// TwinCAT 3 PLC project PLC
// ProgramVersion: 3.1.4026.17
// CompilerDefines: VISU_USEPROPERTYINFO
// libraries:
//   Tc2_Standard, * (Beckhoff Automation GmbH)
//   Tc2_System, * (Beckhoff Automation GmbH)
//   Tc3_Analytics, * (Beckhoff Automation GmbH)
//   TcoCore, * (Vortex.Library)
//   TcoDrivesBeckhoff, * (Vortex.Library)
//   TcoElements, * (Vortex.Library)
//   TcoIo, * (Vortex.Library)
//   TcoPneumatics, * (Vortex.Library)
//   TcoUtilities, * (Vortex.Library)
//   VisuDialogs, * (System)
// project tree:
//   Components/ ST_MachineSetting.TcDUT
//   Components/TcaCarrier/Structures/ TcaCarrierConfig.TcDUT, TcaCarrierService.TcDUT, TcaCarrierData.TcDUT
//   Components/TcaCarrier/Enumerations/ eTcaCarrierCmd.TcDUT (not stored), eTcaCarrierLayout.TcDUT (not stored)
//   Components/TcaCarrier/ ITcaCarrier.TcIO, TcaCarrier.TcPOU
//   Components/TcaCarrier/Tasks/ TcaCarrierModifyTask.TcPOU
//   Components/TcaPushButton/Enumerations/ eTcaPushButtonColor.TcDUT, eTcaPushButtonLightState.TcDUT
//   Components/TcaPushButton/Structures/ TcaPushButtonStatus.TcDUT (not stored), TcaPushButtonRef.TcDUT (not stored), TcaPushButtonConfig.TcDUT (not stored), TcaPushButtonService.TcDUT
//   Components/TcaPushButton/ TcaPushButton.TcPOU
//   Components/TcaStorage/ E_ApproachDirection.TcDUT (not stored), eTcaStorageCmd.TcDUT, TcaRobotStorage.TcPOU (not stored) (excluded from build), TcaStorage.TcPOU, TcaStorageRef.TcDUT
//   Components/TcaTrolley/Structures/ TcaTrolleyData.TcDUT, TcaTrolleyService.TcDUT
//   Components/TcaTrolley/ TcaTrolley.TcPOU
//   Components/TcaTrolley_old/ CMD_Trolley.TcDUT, eTcaTrolleyCmd.TcDUT (not stored), TcaTrolley_old.TcPOU, TcaTrolleyRef.TcDUT (not stored)
//   Components/TcaWorkpiecePlace/Enumerations/ eTcaWorkpiecePlaceStatus.TcDUT, eTcaWorkpiecePlaceShape.TcDUT
//   Components/TcaWorkpiecePlace/Structures/ TcaWorkpiecePlaceService.TcDUT, TcaWorkpiecePlaceData.TcDUT
//   Components/TcaWorkpiecePlace/ TcaWorkpiecePlace.TcPOU
//   Components_RMTH/TcaEngelCasting/ Schnittstellenprotokoll.TcDUT (not stored), TcaEngelCastingCarrierInput.TcDUT (not stored), TcaEngelCastingCarrierJob.TcDUT (not stored), TcaEngelCastingCarrierJobStatus.TcDUT, TcaEngelCastingCarrierOutput.TcDUT (not stored), TcalEngelCastingCarrierStatus.TcDUT (not stored)
//   Components_RMTH/TcaLaserDistanceSenor/Structures/ TcaLaserDistanceSenorConfig.TcDUT (not stored), TcaLaserDistanceSenorRef.TcDUT (not stored), TcaLaserDistanceSenorStatus.TcDUT, TcaLaserDistanceSensorDataArrayEntry.TcDUT (not stored), TcaLaserDistanceSenorService.TcDUT (not stored)
//   Components_RMTH/TcaLaserDistanceSenor/ TcaLaserDistanceSenor.TcPOU (not stored)
//   Components_RMTH/TcaRackFeeder/Structures/ TcaRackFeederConfig.TcDUT (not stored), TcaRackFeederRef.TcDUT (not stored), TcaRackFeederService.TcDUT (not stored), TcaRackFeederStatus.TcDUT
//   Components_RMTH/TcaRackFeeder/ TcaRackFeeder.TcPOU (not stored)
//   Components_RMTH/TcaSafetyGate/ ISafetyComponent.TcIO (not stored), TcaSafetyGate.TcPOU (not stored)
//   Components_RMTH/TcaSafetyGate/Structures/ TcaSafetyGateConfig.TcDUT (not stored), TcaSafetyGateRef.TcDUT, TcaSafetyGateService.TcDUT, TcaSafetyGateStatus.TcDUT
//   Components_RMTH/TcaSegmentDoor/Structures/ TcaSegmentDoorConfig.TcDUT (not stored), TcaSegmentDoorRef.TcDUT (not stored), TcaSegmentDoorService.TcDUT (not stored), TcaSegmentDoorStatus.TcDUT (not stored)
//   Components_RMTH/TcaSegmentDoor/ TcaSegmentDoor.TcPOU
//   Components_RMTH/TcaTwinSAFE/Structures/ TcaTwinSAFEConfig.TcDUT, TcaTwinSAFERef.TcDUT (not stored), TcaTwinSAFEService.TcDUT (not stored), TcaTwinSAFEStatus.TcDUT (not stored)
//   Components_RMTH/TcaTwinSAFE/ TcaTwinSAFE.TcPOU (not stored)
//   / GlobalTextList.TcGTLO, PlcTask.TcTTO, Visualization Manager.TcVMO (not stored)
//   Items/ COLOR.TcDUT, E_Coordinate.TcDUT (not stored), ST_ComboboxEntry.TcDUT, ST_Coordinate.TcDUT (not stored), ST_WorkpieceType.TcDUT
//   Program/Handling/Dialogs/ Handling_TeachRack_DlgContent.TcPOU
//   Program/Handling/Sequences/ Handling_Teach.TcPOU (not stored), Handling_TeachRack.TcPOU (not stored), Handling_GroundMode.TcPOU (not stored), Handling_OpenDoor.TcPOU (not stored)
//   Program/ MAIN.TcPOU, Peripherie.TcPOU
//   Program/Handling/ Handling.TcPOU, Handling_Components.TcPOU (not stored), Handling_Positions.TcPOU (not stored)
//   Template/Component_Cylinder/Base/ CylinderBase.TcPOU, TcoCylinderBase.TcPOU (not stored), TcoDoubleCylinderBase.TcPOU
//   Template/Component_Cylinder/ ITcoCylinder.TcIO (not stored), TcoCylinder.TcPOU, TcoDoubleCylinder.TcPOU
//   Template/Component_Cylinder/Structs/ CylinderConfig.TcDUT, CylinderStatus.TcDUT (not stored), TcoCylinderConfig.TcDUT, TcoCylinderStatus.TcDUT
//   Template/Component_Cylinder/Tasks/ CylinderMoveTask.TcPOU, TcoCylinderMoveTask.TcPOU (not stored)
//   Template/RackFeeder/ CMD_RackFeeder.TcDUT, E_RackFeederCmd.TcDUT (not stored), FB_RackFeeder.TcPOU
//   Template/RackFeeder/Structure/ ST_RackFeederIO.TcDUT, ST_RackFeederJob.TcDUT (not stored), ST_StorageDock.TcDUT (not stored), ST_TrolleyDock.TcDUT (not stored)
//   Template/Station/Data/ ST001_ProcessData.TcDUT (not stored), ST001_ProcessDataManager.TcPOU (not stored)
//   Template/Station/ ST001.TcPOU, ST001_AutomatSequence.TcPOU (not stored), ST001_Components.TcDUT (not stored), ST001_ComponentsHandler.TcPOU, ST001_GroundSequence.TcPOU
//   Template/Component_Carousell/Base/ TcoCarouselBase.TcPOU (not stored)
//   Template/Component_Carousell/Structs/ eTcoCarouselDirection.TcDUT, TcoCarouselConfig.TcDUT, TcoCarouselStatus.TcDUT
//   Template/Component_Carousell/Tasks/ TcoTurnTableTask.TcPOU
//   Template/Component_Carousell/ TcoCarousel.TcPOU (not stored)
//   Utilities/Component/Enumerations/ E_ComponentState.TcDUT, E_SafeState.TcDUT (not stored)
//   Utilities/Component/ FB_Component.TcPOU, FB_ComponentPool.TcPOU (not stored)
//   Utilities/Component/Interfaces/ ITF_Component.TcIO (not stored)
//   Utilities/Component/Structures/ ST_ComponentVisu.TcDUT
//   Utilities/Component/Visualisation/ Uc_Component.TcVIS (not stored)
//   Utilities/EventLog/Base/ FB_LoggingProviderBase.TcPOU (not stored)
//   Utilities/EventLog/Enumerations/ E_BoolFilter.TcDUT (not stored), E_FilterActive.TcDUT (not stored), E_LoggingProvider.TcDUT, E_LogLevel.TcDUT (not stored), E_Priority.TcDUT, ST_LoggingConfig.TcDUT (not stored)
//   Utilities/EventLog/ E_Event.TcDUT, FB_EventLog.TcPOU
//   Utilities/EventLog/Interface/ ITFLoggingProvider.TcIO, ITF_EventLog.TcIO (not stored)
//   Utilities/EventLog/Structures/ ST_Event.TcDUT (not stored), ST_EventBase.TcDUT, ST_EventOutput.TcDUT (not stored), ST_EventVisu.TcDUT, ST_Log.TcDUT (not stored)
//   Utilities/EventLog/Visualization/ Uc_EventLog.TcVIS (not stored), Uc_EventLogControl.TcDUT (not stored), Uc_EventLogControl.TcVIS (not stored), Uc_EventLogEntry.TcVIS (not stored), Uc_EventLogTable.TcDUT (not stored), Uc_EventLogTable.TcVIS (not stored)
//   Utilities/Helpers/Color/ F_DWORD2CMYK.TcPOU (not stored), F_DWORD2RGB.TcPOU, F_RGB2CMYK.TcPOU, F_RGB2DWORD.TcPOU (not stored), F_TextColor.TcPOU, ST_Color.TcDUT (not stored), ST_ColorCMYK.TcDUT
//   Utilities/Helpers/Concat/ Concat10.TcPOU (not stored), Concat2.TcPOU, Concat3.TcPOU (not stored), Concat4.TcPOU (not stored), Concat5.TcPOU (not stored), Concat6.TcPOU (not stored), Concat7.TcPOU, Concat8.TcPOU (not stored), Concat9.TcPOU (not stored), ConcatArray.TcPOU (not stored)
//   Utilities/Helpers/ E_OperationResult.TcDUT, FB_GetTimeString.TcPOU (not stored) (excluded from build), FB_Pulse.TcPOU (not stored), FB_TON_RMTH.TcPOU (not stored), F_BYTE_TO_INT.TcPOU (not stored), F_BYTE_TO_REAL.TcPOU, F_DT_TO_STRING.TcPOU, F_GetAdsPort.TcPOU, F_GetPlcCycleTime.TcPOU (not stored), F_GetSystemTime64.TcPOU (not stored), F_TO_STRING.TcPOU (not stored), P_FilePath.TcPOU, P_System.TcPOU (not stored), ST_DefaultPulse.TcDUT, ST_PlcSystemInfo.TcDUT
//   Utilities/ HexColor.TcGVL (not stored), Statics.TcGVL (not stored), StaticsConstant.TcGVL
//   Utilities/List/ FB_List.TcPOU
//   Utilities/List/Structures/ ST_Listentry.TcDUT, Uc_List.TcDUT (not stored)
//   Utilities/List/Visu/ Uc_EntryDetail.TcVIS, Uc_List.TcVIS (not stored), Uc_Listentry.TcVIS (not stored)
//   Utilities/Sequencer/Enumeration/ E_SequenceState.TcDUT (not stored)
//   Utilities/Sequencer/ FB_Sequence.TcPOU (not stored)
// real-time tasks:
//   TASK PlcTask: cycle T#10ms, priority 20, ADS port 350
// motion (NC):
//   TASK NC-Task 1 SAF: cycle T#2ms, priority 4, ADS port 501
//   TASK NC-Task 1 SVB: cycle T#10ms, priority 8, ADS port 511
//   AXIS Oven B CH1 (id 14)
//     Dynamic: Acceleration=282800000, Deceleration=282800000, Jerk=2.85628e+17
//     Velo: RefSearch=25, RefSync=25, SlowManual=14, FastManual=28, Maximum=28
//     PositionAreaControl: Enable=false
//     TargetPosControl: Enable=false
//     OtherSettings: AllowMotionCmdToSlave=true
//     encoder EncType=7
//       EncPara: ScaleFactorNumerator=0.001879, Offset=-1.4, MaxCount=#x0000ffff, ReferenceSystem=1
//     drive DrvType=23
//       Analog: VeloReferenz=28, TorqueSetpointScale=10, ScaleFactorActTorque=0.1
//       TimeComp: TaskDelayCycles=1
//     controller CtrType=1
//       CtrPara: PriorControlFactor=1
//         PosDiffControl: Enable=false
//         Observer: BandWidth=20
//   AXIS Storage A (id 2)
//     Dynamic: Acceleration=282800000, Deceleration=282800000, Jerk=2.85628e+17
//     Velo: RefSearch=25, RefSync=25, SlowManual=14, FastManual=28, Maximum=28
//     PositionAreaControl: Enable=false
//     TargetPosControl: Enable=false
//     OtherSettings: AllowMotionCmdToSlave=true
//     encoder EncType=1
//       EncPara: ScaleFactorNumerator=0.00751766651631334, Offset=-1.4
//     drive DrvType=23
//       Analog: VeloReferenz=28, TorqueSetpointScale=10, ScaleFactorActTorque=0.1
//       TimeComp: TaskDelayCycles=1
//     controller CtrType=1
//       CtrPara: PriorControlFactor=1
//         PosDiffControl: Enable=false
//         Observer: BandWidth=20
//   AXIS Oven B CH2 (id 15)
//     Dynamic: Acceleration=282800000, Deceleration=282800000, Jerk=2.85628e+17
//     Velo: RefSearch=25, RefSync=25, SlowManual=14, FastManual=28, Maximum=28
//     PositionAreaControl: Enable=false
//     TargetPosControl: Enable=false
//     OtherSettings: AllowMotionCmdToSlave=true
//     encoder EncType=7
//       EncPara: ScaleFactorNumerator=0.001879, Offset=-1.4, MaxCount=#x0000ffff, ReferenceSystem=1
//     drive DrvType=23
//       Analog: VeloReferenz=28, TorqueSetpointScale=10, ScaleFactorActTorque=0.1
//       TimeComp: TaskDelayCycles=1
//     controller CtrType=1
//       CtrPara: PriorControlFactor=1
//         PosDiffControl: Enable=false
//         Observer: BandWidth=20
//   AXIS Rackfeeder X (id 16)
//     Dynamic: Acceleration=2461.9275, Deceleration=2461.9275, Jerk=7385.7825
//     Velo: RefSearch=16.41285, RefSync=16.41285, SlowManual=10, FastManual=60, Fast=1641.285, Maximum=1641.285
//     OtherSettings: AllowMotionCmdToSlave=true
//     encoder EncType=8
//       EncPara: ScaleFactorNumerator=150, ScaleFactorDenominator=10485760, MaxCount=#xffffffff
//     drive DrvType=9
//       DrvPara: MaxCount=#xffffffff, DriveControlDWord=#x00030100
//         Analog: VeloReferenz=1805.4135, VeloScale=1.02400649589962, TorqueSetpointScale=10, ScaleFactorActTorque=0.1
//         TimeComp: TaskDelayCycles=1
//     controller CtrType=1
//       CtrPara: PriorControlFactor=1
//         Observer: BandWidth=20
//   AXIS Rackfeeder Y (id 17)
//     Dynamic: Acceleration=2256.7665, Deceleration=2256.7665, Jerk=6770.2995
//     Velo: RefSearch=15.04511, RefSync=15.04511, SlowManual=10, FastManual=60, Fast=1504.511, Maximum=1504.511
//     OtherSettings: AllowMotionCmdToSlave=true
//     encoder EncType=8
//       EncPara: ScaleFactorNumerator=220, ScaleFactorDenominator=16777216, MaxCount=#xffffffff
//     drive DrvType=9
//       DrvPara: MaxCount=#xffffffff, DriveControlDWord=#x00030100
//         Analog: VeloReferenz=1654.9621, VeloScale=1.02400649589962, TorqueSetpointScale=10, ScaleFactorActTorque=0.1
//         TimeComp: TaskDelayCycles=1
//     controller CtrType=1
//       CtrPara: PriorControlFactor=1
//         Observer: BandWidth=20
//   AXIS Rackfeeder Teleskop (id 18)
//     OtherSettings: AllowMotionCmdToSlave=true
//     encoder EncType=8
//       EncPara: MaxCount=#xffffffff
//     drive DrvType=9
//       DrvPara: MaxCount=#xffffffff, DriveControlDWord=#x00030100
//         Analog: VeloScale=1.02400649589962, TorqueSetpointScale=10, ScaleFactorActTorque=0.1
//         TimeComp: TaskDelayCycles=1
//     controller CtrType=1
//       CtrPara: PriorControlFactor=1
//         Observer: BandWidth=20
//   AXIS Oven B (id 21)
//     Dynamic: Acceleration=1231.0125, Deceleration=1231.0125, Jerk=3693.0375
//     Velo: RefSearch=8.20675, RefSync=8.20675, SlowManual=20, FastManual=120, Fast=820.675, Maximum=820.675
//     OtherSettings: AllowMotionCmdToSlave=true
//     encoder EncType=8
//       EncPara: ScaleFactorNumerator=120, ScaleFactorDenominator=16777216, Inverse=true, MaxCount=#xffffffff
//     drive DrvType=9
//       DrvPara: Inverse=true, MaxCount=#xffffffff, DriveControlDWord=#x00030100
//         Analog: VeloReferenz=902.7425, VeloScale=1.02400649589962, TorqueSetpointScale=10, ScaleFactorActTorque=0.1
//         TimeComp: TaskDelayCycles=1
//     controller CtrType=1
//       CtrPara: PriorControlFactor=1
//         Observer: BandWidth=20
//   AXIS Oven A (id 20)
//     Dynamic: Acceleration=1231.0125, Deceleration=1231.0125, Jerk=3693.0375
//     Velo: RefSearch=8.20675, RefSync=8.20675, SlowManual=20, FastManual=120, Fast=820.675, Maximum=820.675
//     OtherSettings: AllowMotionCmdToSlave=true
//     encoder EncType=8
//       EncPara: ScaleFactorNumerator=120, ScaleFactorDenominator=16777216, Inverse=true, MaxCount=#xffffffff
//     drive DrvType=9
//       DrvPara: Inverse=true, MaxCount=#xffffffff, DriveControlDWord=#x00030100
//         Analog: VeloReferenz=902.7425, VeloScale=1.02400649589962, TorqueSetpointScale=10, ScaleFactorActTorque=0.1
//         TimeComp: TaskDelayCycles=1
//     controller CtrType=1
//       CtrPara: PriorControlFactor=1
//         Observer: BandWidth=20
//   AXIS Oven A CH1 (id 1)
//     Dynamic: Acceleration=282800000, Deceleration=282800000, Jerk=2.85628e+17, DelayTime=0.01, OverrideType=4
//     Velo: RefSearch=25, RefSync=25, SlowManual=14, FastManual=28, Maximum=28
//     PositionAreaControl: Enable=false
//     TargetPosControl: Enable=false
//     OtherSettings: AllowMotionCmdToSlave=true
//     encoder EncType=7
//       EncPara: ScaleFactorNumerator=0.001879, Offset=-1.4, EncMode=1, MaxCount=#x0000ffff, ReferenceSystem=1
//         FilterTime: TVelo=0.1
//         SoftEndMinControl: Range=-5
//         SoftEndMaxControl: Range=30
//         ActPosCorrection: Enable=true, Time=1
//     drive DrvType=23
//       Analog: VeloReferenz=28, TorqueSetpointScale=10, ScaleFactorActTorque=0.1
//       TimeComp: TaskDelayCycles=1
//     controller CtrType=1
//       CtrPara: PriorControlFactor=1
//         PosDiffControl: Enable=false
//         Observer: BandWidth=20
//   AXIS Oven A CH2 (id 13)
//     Dynamic: Acceleration=282800000, Deceleration=282800000, Jerk=2.85628e+17
//     Velo: RefSearch=25, RefSync=25, SlowManual=14, FastManual=28, Maximum=28
//     PositionAreaControl: Enable=false
//     TargetPosControl: Enable=false
//     OtherSettings: AllowMotionCmdToSlave=true
//     encoder EncType=7
//       EncPara: ScaleFactorNumerator=0.001879, Offset=-1.4, MaxCount=#x0000ffff, ReferenceSystem=1
//     drive DrvType=23
//       Analog: VeloReferenz=28, TorqueSetpointScale=10, ScaleFactorActTorque=0.1
//       TimeComp: TaskDelayCycles=1
//     controller CtrType=1
//       CtrPara: PriorControlFactor=1
//         PosDiffControl: Enable=false
//         Observer: BandWidth=20
//   AXIS Storage B (id 3)
//     Dynamic: Acceleration=282800000, Deceleration=282800000, Jerk=2.85628e+17
//     Velo: RefSearch=25, RefSync=25, SlowManual=14, FastManual=28, Maximum=28
//     PositionAreaControl: Enable=false
//     TargetPosControl: Enable=false
//     OtherSettings: AllowMotionCmdToSlave=true
//     encoder EncType=1
//       EncPara: ScaleFactorNumerator=0.00751766651631334, Offset=-1.4
//     drive DrvType=23
//       Analog: VeloReferenz=28, TorqueSetpointScale=10, ScaleFactorActTorque=0.1
//       TimeComp: TaskDelayCycles=1
//     controller CtrType=1
//       CtrPara: PriorControlFactor=1
//         PosDiffControl: Enable=false
//         Observer: BandWidth=20
// I/O:
//   DEVICE Gerät 3 (EtherCAT) (disabled), AmsNetId 41.249.230.93.4.1
//     Klemme 1 (EK1100) [EK1100 EtherCAT-Koppler (2A E-Bus)]
//       Klemme 33 (EL6910) [EL6910, TwinSAFE PLC]
//       Klemme 3 (EL1904) [EL1904, 4 K. Safety Eingang 24V, TwinSAFE]
//         modules: Module 1 (FSOES)
//       Klemme 4 (EL2904) [EL2904, 4 K. Safety Ausgang 24V, 0.5A, TwinSAFE]
//         modules: Module 1 (FSOES), Module 2 (DO)
//       Klemme 5 (EL1104) [EL1104 4K. Dig. Eingang 24V, 3ms, Sensorversorgung]
//       Klemme 6 (EL1104) [EL1104 4K. Dig. Eingang 24V, 3ms, Sensorversorgung]
//       Klemme 7 (EL6224) [EL6224 (IO Link Master)]
//       ENGEL Interface (EL1008) [EL1008 8K. Dig. Eingang 24V, 3ms]
//       ENGEL Interface (EL2624) [EL2624 4K. Relais Ausgang, Schließer (125V AC / 30V DC)]
//       Ovens (EK1122) [EK1122 2-Port EtherCAT-Abzweig]
//         Oven_A (EK1100) [EK1100 EtherCAT-Koppler (2A E-Bus)]
//           Klemme 10 (EL1904) [EL1904, 4 K. Safety Eingang 24V, TwinSAFE]
//             modules: Module 1 (FSOES)
//           Klemme 11 (EL2904) [EL2904, 4 K. Safety Ausgang 24V, 0.5A, TwinSAFE]
//             modules: Module 1 (FSOES), Module 2 (DO)
//           Klemme 12 (EL7332) [EL7332 2K. DC-Motor-Endstufe (24V, 1.5A)]
//           Klemme 13 (EL3062-0030) [EL3062-0030 2K.Ana. Eingang 0-30V]
//           Klemme 14 (EL1004) [EL1004 4K. Dig. Eingang 24V, 3ms]
//           Klemme 15 (EL2004) [EL2004 4K. Dig. Ausgang 24V, 0.5A]
//           Klemme 16 (EL9010) [EL9010 Endklemme]
//         Oven_B (EK1100) [EK1100 EtherCAT-Koppler (2A E-Bus)]
//           Klemme 18 (EL1904) [EL1904, 4 K. Safety Eingang 24V, TwinSAFE]
//             modules: Module 1 (FSOES)
//           Klemme 19 (EL2904) [EL2904, 4 K. Safety Ausgang 24V, 0.5A, TwinSAFE]
//             modules: Module 1 (FSOES), Module 2 (DO)
//           Klemme 20 (EL7332) [EL7332 2K. DC-Motor-Endstufe (24V, 1.5A)]
//           Klemme 21 (EL3062-0030) [EL3062-0030 2K.Ana. Eingang 0-30V]
//           Klemme 22 (EL1004) [EL1004 4K. Dig. Eingang 24V, 3ms]
//           Klemme 23 (EL2004) [EL2004 4K. Dig. Ausgang 24V, 0.5A]
//           Klemme 61 (EL9010) [EL9010 Endklemme]
//       Storage|Casting (EK1122) [EK1122 2-Port EtherCAT-Abzweig]
//         Storage (EK1100)
//     RackFeeder_X_Y (AX5206-0000-0215) [AX5206-0000-0215 EtherCAT Drive (SoE, 2 Ch.)]
//       Klemme 27 (AX5805) [AX5805 (Safety Drive Option)]
//         modules: Module 1 (Safety Process Data, 2 axis), Module 2 (Standard Process Data, 2 axis)
//     Rackfeeder_Teleskop (AX5203-0000-0215) [AX5203-0000-0215 EtherCAT Drive (SoE, 2 Ch.)]
//       Klemme 29 (AX5805) [AX5805 (Safety Drive Option)]
//         modules: Module 1 (Safety Process Data, 2 axis), Module 2 (Standard Process Data, 2 axis)
//     OvenDoor_A_B (AX5206-0000-0215) [AX5206-0000-0215 EtherCAT Drive (SoE, 2 Ch.)]
//       Klemme 31 (AX5805) [AX5805 (Safety Drive Option)]
//         modules: Module 1 (Safety Process Data, 2 axis), Module 2 (Standard Process Data, 2 axis)
// variable links:
//   Device 3 (EtherCAT) <-> Device 3 (EtherCAT)/OvenDoor_A_B (AX5206-0000-0215)/Term 31 (AX5805)
//     Term 1 (EK1100)/Term 33 (EL6910)/ConnectionInputs/TwinSafeMain.Oven (AX5805) - Module 1 (Safety Process Data, 2 axis)_120 TxPDO <-> Module 1 (Safety Process Data, 2 axis)/Outputs (Controlword)/FSOE
//     Term 1 (EK1100)/Term 33 (EL6910)/ConnectionOutputs/TwinSafeMain.Oven (AX5805) - Module 1 (Safety Process Data, 2 axis)_120 RxPDO <-> Module 1 (Safety Process Data, 2 axis)/Inputs (Statusword)/FSOE
//   Device 3 (EtherCAT) <-> Device 3 (EtherCAT)/RackFeeder_X_Y (AX5206-0000-0215)/Term 27 (AX5805)
//     Term 1 (EK1100)/Term 33 (EL6910)/ConnectionInputs/TwinSafeMain.Rackfeeder_XY (AX5805) - Module 1 (Safety Process Data, 2 axis)_118 TxPDO <-> Module 1 (Safety Process Data, 2 axis)/Outputs (Controlword)/FSOE
//     Term 1 (EK1100)/Term 33 (EL6910)/ConnectionOutputs/TwinSafeMain.Rackfeeder_XY (AX5805) - Module 1 (Safety Process Data, 2 axis)_118 RxPDO <-> Module 1 (Safety Process Data, 2 axis)/Inputs (Statusword)/FSOE
//   Device 3 (EtherCAT) <-> Device 3 (EtherCAT)/Rackfeeder_Teleskop (AX5203-0000-0215)/Term 29 (AX5805)
//     Term 1 (EK1100)/Term 33 (EL6910)/ConnectionInputs/TwinSafeMain.Rackfeeder_Tele (AX5805) - Module 1 (Safety Process Data, 2 axis)_119 TxPDO <-> Module 1 (Safety Process Data, 2 axis)/Outputs (Controlword)/FSOE
//     Term 1 (EK1100)/Term 33 (EL6910)/ConnectionOutputs/TwinSafeMain.Rackfeeder_Tele (AX5805) - Module 1 (Safety Process Data, 2 axis)_119 RxPDO <-> Module 1 (Safety Process Data, 2 axis)/Inputs (Statusword)/FSOE
//   Device 3 (EtherCAT) <-> Device 3 (EtherCAT)/Term 1 (EK1100)/Ovens (EK1122)/Oven_A (EK1100)/Term 10 (EL1904)
//     Term 1 (EK1100)/Term 33 (EL6910)/ConnectionInputs/TwinSafeMain.Oven A (EL1904) - Module 1 (FSOES)_14 TxPDO <-> Module 1 (FSOES)/RxPDO/FSOE
//     Term 1 (EK1100)/Term 33 (EL6910)/ConnectionOutputs/TwinSafeMain.Oven A (EL1904) - Module 1 (FSOES)_14 RxPDO <-> Module 1 (FSOES)/TxPDO/FSOE
//   Device 3 (EtherCAT) <-> Device 3 (EtherCAT)/Term 1 (EK1100)/Ovens (EK1122)/Oven_A (EK1100)/Term 11 (EL2904)
//     Term 1 (EK1100)/Term 33 (EL6910)/ConnectionInputs/TwinSafeMain.Oven A (EL2904) - Module 1 (FSOES)_111 TxPDO <-> Module 1 (FSOES)/RxPDO/FSOE
//     Term 1 (EK1100)/Term 33 (EL6910)/ConnectionOutputs/TwinSafeMain.Oven A (EL2904) - Module 1 (FSOES)_111 RxPDO <-> Module 1 (FSOES)/TxPDO/FSOE
//   Device 3 (EtherCAT) <-> Device 3 (EtherCAT)/Term 1 (EK1100)/Ovens (EK1122)/Oven_B (EK1100)/Term 18 (EL1904)
//     Term 1 (EK1100)/Term 33 (EL6910)/ConnectionInputs/TwinSafeMain.Oven B (EL1904) - Module 1 (FSOES)_16 TxPDO <-> Module 1 (FSOES)/RxPDO/FSOE
//     Term 1 (EK1100)/Term 33 (EL6910)/ConnectionOutputs/TwinSafeMain.Oven B (EL1904) - Module 1 (FSOES)_16 RxPDO <-> Module 1 (FSOES)/TxPDO/FSOE
//   Device 3 (EtherCAT) <-> Device 3 (EtherCAT)/Term 1 (EK1100)/Ovens (EK1122)/Oven_B (EK1100)/Term 19 (EL2904)
//     Term 1 (EK1100)/Term 33 (EL6910)/ConnectionInputs/TwinSafeMain.Oven B (EL2904) - Module 1 (FSOES)_112 TxPDO <-> Module 1 (FSOES)/RxPDO/FSOE
//     Term 1 (EK1100)/Term 33 (EL6910)/ConnectionOutputs/TwinSafeMain.Oven B (EL2904) - Module 1 (FSOES)_112 RxPDO <-> Module 1 (FSOES)/TxPDO/FSOE
//   Device 3 (EtherCAT) <-> Device 3 (EtherCAT)/Term 1 (EK1100)/Term 3 (EL1904)
//     Term 1 (EK1100)/Term 33 (EL6910)/ConnectionInputs/TwinSafeMain.MAIN (EL1904) - Module 1 (FSOES)_12 TxPDO <-> Module 1 (FSOES)/RxPDO/FSOE
//     Term 1 (EK1100)/Term 33 (EL6910)/ConnectionOutputs/TwinSafeMain.MAIN (EL1904) - Module 1 (FSOES)_12 RxPDO <-> Module 1 (FSOES)/TxPDO/FSOE
//   Device 3 (EtherCAT) <-> Device 3 (EtherCAT)/Term 1 (EK1100)/Term 4 (EL2904)
//     Term 1 (EK1100)/Term 33 (EL6910)/ConnectionInputs/TwinSafeMain.MAIN (EL2904) - Module 1 (FSOES)_13 TxPDO <-> Module 1 (FSOES)/RxPDO/FSOE
//     Term 1 (EK1100)/Term 33 (EL6910)/ConnectionOutputs/TwinSafeMain.MAIN (EL2904) - Module 1 (FSOES)_13 RxPDO <-> Module 1 (FSOES)/TxPDO/FSOE
//   NC-Task 1 SAF/Axes/Oven A <-> Device 3 (EtherCAT)/OvenDoor_A_B (AX5206-0000-0215)
//     Drive/Inputs/In/nDataIn1 <-> AT 1/Following distance
//     Drive/Inputs/In/nDcOutputTime <-> InfoData/DcOutputShift
//     Drive/Inputs/In/nState1 <-> AT 1/Drive status word @bit 8
//     Drive/Inputs/In/nState2 <-> AT 1/Drive status word
//     Drive/Inputs/In/nState4 @bit 1 <-> WcState/InputToggle
//     Drive/Inputs/In/nState4 <-> WcState/WcState
//     Drive/Outputs/Out/nCtrl1 <-> MDT 1/Master control word @bit 8
//     Drive/Outputs/Out/nDataOut1 <-> MDT 1/Position command value
//     Enc/Inputs/In/nDataIn1 <-> AT 1/Position feedback 1 value
//     Enc/Inputs/In/nDcInputTime <-> InfoData/DcInputShift
//     Enc/Inputs/In/nState4 @bit 1 <-> WcState/InputToggle
//     Enc/Inputs/In/nState4 <-> WcState/WcState
//   NC-Task 1 SAF/Axes/Oven A CH1 <-> Device 3 (EtherCAT)/Term 1 (EK1100)/Ovens (EK1122)/Oven_A (EK1100)/Term 12 (EL7332)
//     Drive/Inputs/In/nState1 @bit 3 <-> DCM Status Channel 1/Status/Error
//     Drive/Inputs/In/nState1 @bit 5 <-> DCM Status Channel 1/Status/Moving negative
//     Drive/Inputs/In/nState1 @bit 4 <-> DCM Status Channel 1/Status/Moving positive
//     Drive/Inputs/In/nState1 @bit 1 <-> DCM Status Channel 1/Status/Ready
//     Drive/Inputs/In/nState1 <-> DCM Status Channel 1/Status/Ready to enable
//     Drive/Inputs/In/nState1 @bit 6 <-> DCM Status Channel 1/Status/Torque reduced
//     Drive/Inputs/In/nState1 @bit 2 <-> DCM Status Channel 1/Status/Warning
//     Drive/Inputs/In/nState2 @bit 3 <-> DCM Status Channel 1/Status/Digital input 1
//     Drive/Inputs/In/nState2 @bit 4 <-> DCM Status Channel 1/Status/Digital input 2
//     Drive/Inputs/In/nState2 @bit 5 <-> DCM Status Channel 1/Status/Sync error
//     Drive/Inputs/In/nState2 @bit 7 <-> DCM Status Channel 1/Status/TxPDO Toggle
//     Drive/Inputs/In/nState4 @bit 1 <-> WcState/InputToggle
//     Drive/Inputs/In/nState4 <-> WcState/WcState
//     Drive/Outputs/Out/nCtrl1 <-> DCM Control Channel 1/Control/Enable
//     Drive/Outputs/Out/nCtrl1 @bit 2 <-> DCM Control Channel 1/Control/Reduce torque
//     Drive/Outputs/Out/nCtrl1 @bit 1 <-> DCM Control Channel 1/Control/Reset
//     Drive/Outputs/Out/nDataOut2[0] <-> DCM Velocity Channel 1/Velocity
//   NC-Task 1 SAF/Axes/Oven A CH1 <-> Device 3 (EtherCAT)/Term 1 (EK1100)/Ovens (EK1122)/Oven_A (EK1100)/Term 13 (EL3062-0030)
//     Enc/Inputs/In/nDataIn1[0] <-> AI Standard Channel 1/Value
//     Enc/Inputs/In/nState4 @bit 1 <-> WcState/InputToggle
//     Enc/Inputs/In/nState4 <-> WcState/WcState
//   NC-Task 1 SAF/Axes/Oven A CH2 <-> Device 3 (EtherCAT)/Term 1 (EK1100)/Ovens (EK1122)/Oven_A (EK1100)/Term 12 (EL7332)
//     Drive/Inputs/In/nState1 @bit 3 <-> DCM Status Channel 2/Status/Error
//     Drive/Inputs/In/nState1 @bit 5 <-> DCM Status Channel 2/Status/Moving negative
//     Drive/Inputs/In/nState1 @bit 4 <-> DCM Status Channel 2/Status/Moving positive
//     Drive/Inputs/In/nState1 @bit 1 <-> DCM Status Channel 2/Status/Ready
//     Drive/Inputs/In/nState1 <-> DCM Status Channel 2/Status/Ready to enable
//     Drive/Inputs/In/nState1 @bit 6 <-> DCM Status Channel 2/Status/Torque reduced
//     Drive/Inputs/In/nState1 @bit 2 <-> DCM Status Channel 2/Status/Warning
//     Drive/Inputs/In/nState2 @bit 3 <-> DCM Status Channel 2/Status/Digital input 1
//     Drive/Inputs/In/nState2 @bit 4 <-> DCM Status Channel 2/Status/Digital input 2
//     Drive/Inputs/In/nState2 @bit 5 <-> DCM Status Channel 2/Status/Sync error
//     Drive/Inputs/In/nState2 @bit 7 <-> DCM Status Channel 2/Status/TxPDO Toggle
//     Drive/Inputs/In/nState4 @bit 1 <-> WcState/InputToggle
//     Drive/Inputs/In/nState4 <-> WcState/WcState
//     Drive/Outputs/Out/nCtrl1 <-> DCM Control Channel 2/Control/Enable
//     Drive/Outputs/Out/nCtrl1 @bit 2 <-> DCM Control Channel 2/Control/Reduce torque
//     Drive/Outputs/Out/nCtrl1 @bit 1 <-> DCM Control Channel 2/Control/Reset
//     Drive/Outputs/Out/nDataOut2[0] <-> DCM Velocity Channel 2/Velocity
//   NC-Task 1 SAF/Axes/Oven A CH2 <-> Device 3 (EtherCAT)/Term 1 (EK1100)/Ovens (EK1122)/Oven_A (EK1100)/Term 13 (EL3062-0030)
//     Enc/Inputs/In/nDataIn1[0] <-> AI Standard Channel 2/Value
//     Enc/Inputs/In/nState4 @bit 1 <-> WcState/InputToggle
//     Enc/Inputs/In/nState4 <-> WcState/WcState
//   NC-Task 1 SAF/Axes/Oven B <-> Device 3 (EtherCAT)/OvenDoor_A_B (AX5206-0000-0215)
//     Drive/Inputs/In/nDataIn1 <-> AT 2/Following distance
//     Drive/Inputs/In/nDcOutputTime <-> InfoData/DcOutputShift
//     Drive/Inputs/In/nState1 <-> AT 2/Drive status word @bit 8
//     Drive/Inputs/In/nState2 <-> AT 2/Drive status word
//     Drive/Inputs/In/nState4 @bit 1 <-> WcState/InputToggle
//     Drive/Inputs/In/nState4 <-> WcState/WcState
//     Drive/Outputs/Out/nCtrl1 <-> MDT 2/Master control word @bit 8
//     Drive/Outputs/Out/nDataOut1 <-> MDT 2/Position command value
//     Enc/Inputs/In/nDataIn1 <-> AT 2/Position feedback 1 value
//     Enc/Inputs/In/nDcInputTime <-> InfoData/DcInputShift
//     Enc/Inputs/In/nState4 @bit 1 <-> WcState/InputToggle
//     Enc/Inputs/In/nState4 <-> WcState/WcState
//   NC-Task 1 SAF/Axes/Oven B CH1 <-> Device 3 (EtherCAT)/Term 1 (EK1100)/Ovens (EK1122)/Oven_B (EK1100)/Term 20 (EL7332)
//     Drive/Inputs/In/nState1 @bit 3 <-> DCM Status Channel 1/Status/Error
//     Drive/Inputs/In/nState1 @bit 5 <-> DCM Status Channel 1/Status/Moving negative
//     Drive/Inputs/In/nState1 @bit 4 <-> DCM Status Channel 1/Status/Moving positive
//     Drive/Inputs/In/nState1 @bit 1 <-> DCM Status Channel 1/Status/Ready
//     Drive/Inputs/In/nState1 <-> DCM Status Channel 1/Status/Ready to enable
//     Drive/Inputs/In/nState1 @bit 6 <-> DCM Status Channel 1/Status/Torque reduced
//     Drive/Inputs/In/nState1 @bit 2 <-> DCM Status Channel 1/Status/Warning
//     Drive/Inputs/In/nState2 @bit 3 <-> DCM Status Channel 1/Status/Digital input 1
//     Drive/Inputs/In/nState2 @bit 4 <-> DCM Status Channel 1/Status/Digital input 2
//     Drive/Inputs/In/nState2 @bit 5 <-> DCM Status Channel 1/Status/Sync error
//     Drive/Inputs/In/nState2 @bit 7 <-> DCM Status Channel 1/Status/TxPDO Toggle
//     Drive/Inputs/In/nState4 @bit 1 <-> WcState/InputToggle
//     Drive/Inputs/In/nState4 <-> WcState/WcState
//     Drive/Outputs/Out/nCtrl1 <-> DCM Control Channel 1/Control/Enable
//     Drive/Outputs/Out/nCtrl1 @bit 2 <-> DCM Control Channel 1/Control/Reduce torque
//     Drive/Outputs/Out/nCtrl1 @bit 1 <-> DCM Control Channel 1/Control/Reset
//     Drive/Outputs/Out/nDataOut2[0] <-> DCM Velocity Channel 1/Velocity
//   NC-Task 1 SAF/Axes/Oven B CH1 <-> Device 3 (EtherCAT)/Term 1 (EK1100)/Ovens (EK1122)/Oven_B (EK1100)/Term 21 (EL3062-0030)
//     Enc/Inputs/In/nDataIn1[0] <-> AI Standard Channel 1/Value
//     Enc/Inputs/In/nState4 @bit 1 <-> WcState/InputToggle
//     Enc/Inputs/In/nState4 <-> WcState/WcState
//   NC-Task 1 SAF/Axes/Oven B CH2 <-> Device 3 (EtherCAT)/Term 1 (EK1100)/Ovens (EK1122)/Oven_B (EK1100)/Term 20 (EL7332)
//     Drive/Inputs/In/nState1 @bit 3 <-> DCM Status Channel 2/Status/Error
//     Drive/Inputs/In/nState1 @bit 5 <-> DCM Status Channel 2/Status/Moving negative
//     Drive/Inputs/In/nState1 @bit 4 <-> DCM Status Channel 2/Status/Moving positive
//     Drive/Inputs/In/nState1 @bit 1 <-> DCM Status Channel 2/Status/Ready
//     Drive/Inputs/In/nState1 <-> DCM Status Channel 2/Status/Ready to enable
//     Drive/Inputs/In/nState1 @bit 6 <-> DCM Status Channel 2/Status/Torque reduced
//     Drive/Inputs/In/nState1 @bit 2 <-> DCM Status Channel 2/Status/Warning
//     Drive/Inputs/In/nState2 @bit 3 <-> DCM Status Channel 2/Status/Digital input 1
//     Drive/Inputs/In/nState2 @bit 4 <-> DCM Status Channel 2/Status/Digital input 2
//     Drive/Inputs/In/nState2 @bit 5 <-> DCM Status Channel 2/Status/Sync error
//     Drive/Inputs/In/nState2 @bit 7 <-> DCM Status Channel 2/Status/TxPDO Toggle
//     Drive/Inputs/In/nState4 @bit 1 <-> WcState/InputToggle
//     Drive/Inputs/In/nState4 <-> WcState/WcState
//     Drive/Outputs/Out/nCtrl1 <-> DCM Control Channel 2/Control/Enable
//     Drive/Outputs/Out/nCtrl1 @bit 2 <-> DCM Control Channel 2/Control/Reduce torque
//     Drive/Outputs/Out/nCtrl1 @bit 1 <-> DCM Control Channel 2/Control/Reset
//     Drive/Outputs/Out/nDataOut2[0] <-> DCM Velocity Channel 2/Velocity
//   NC-Task 1 SAF/Axes/Oven B CH2 <-> Device 3 (EtherCAT)/Term 1 (EK1100)/Ovens (EK1122)/Oven_B (EK1100)/Term 21 (EL3062-0030)
//     Enc/Inputs/In/nDataIn1[0] <-> AI Standard Channel 2/Value
//     Enc/Inputs/In/nState4 @bit 1 <-> WcState/InputToggle
//     Enc/Inputs/In/nState4 <-> WcState/WcState
//   NC-Task 1 SAF/Axes/Rackfeeder Teleskop <-> Device 3 (EtherCAT)/Rackfeeder_Teleskop (AX5203-0000-0215)
//     Drive/Inputs/In/nDataIn1 <-> AT 1/Following distance
//     Drive/Inputs/In/nDcOutputTime <-> InfoData/DcOutputShift
//     Drive/Inputs/In/nState1 <-> AT 1/Drive status word @bit 8
//     Drive/Inputs/In/nState2 <-> AT 1/Drive status word
//     Drive/Inputs/In/nState4 @bit 1 <-> WcState/InputToggle
//     Drive/Inputs/In/nState4 <-> WcState/WcState
//     Drive/Outputs/Out/nCtrl1 <-> MDT 1/Master control word @bit 8
//     Drive/Outputs/Out/nDataOut1 <-> MDT 1/Position command value
//     Enc/Inputs/In/nDataIn1 <-> AT 1/Position feedback 1 value
//     Enc/Inputs/In/nDcInputTime <-> InfoData/DcInputShift
//     Enc/Inputs/In/nState4 @bit 1 <-> WcState/InputToggle
//     Enc/Inputs/In/nState4 <-> WcState/WcState
//   NC-Task 1 SAF/Axes/Rackfeeder X <-> Device 3 (EtherCAT)/RackFeeder_X_Y (AX5206-0000-0215)
//     Drive/Inputs/In/nDataIn1 <-> AT 1/Following distance
//     Drive/Inputs/In/nDcOutputTime <-> InfoData/DcOutputShift
//     Drive/Inputs/In/nState1 <-> AT 1/Drive status word @bit 8
//     Drive/Inputs/In/nState2 <-> AT 1/Drive status word
//     Drive/Inputs/In/nState4 @bit 1 <-> WcState/InputToggle
//     Drive/Inputs/In/nState4 <-> WcState/WcState
//     Drive/Outputs/Out/nCtrl1 <-> MDT 1/Master control word @bit 8
//     Drive/Outputs/Out/nDataOut1 <-> MDT 1/Position command value
//     Enc/Inputs/In/nDataIn1 <-> AT 1/Position feedback 1 value
//     Enc/Inputs/In/nDcInputTime <-> InfoData/DcInputShift
//     Enc/Inputs/In/nState4 @bit 1 <-> WcState/InputToggle
//     Enc/Inputs/In/nState4 <-> WcState/WcState
//   NC-Task 1 SAF/Axes/Rackfeeder Y <-> Device 3 (EtherCAT)/RackFeeder_X_Y (AX5206-0000-0215)
//     Drive/Inputs/In/nDataIn1 <-> AT 2/Following distance
//     Drive/Inputs/In/nDcOutputTime <-> InfoData/DcOutputShift
//     Drive/Inputs/In/nState1 <-> AT 2/Drive status word @bit 8
//     Drive/Inputs/In/nState2 <-> AT 2/Drive status word
//     Drive/Inputs/In/nState4 @bit 1 <-> WcState/InputToggle
//     Drive/Inputs/In/nState4 <-> WcState/WcState
//     Drive/Outputs/Out/nCtrl1 <-> MDT 2/Master control word @bit 8
//     Drive/Outputs/Out/nDataOut1 <-> MDT 2/Position command value
//     Enc/Inputs/In/nDataIn1 <-> AT 2/Position feedback 1 value
//     Enc/Inputs/In/nDcInputTime <-> InfoData/DcInputShift
//     Enc/Inputs/In/nState4 @bit 1 <-> WcState/InputToggle
//     Enc/Inputs/In/nState4 <-> WcState/WcState
//   NC-Task 1 SAF/Axes/Storage A <-> Device 3 (EtherCAT)/Term 1 (EK1100)/Storage|Casting (EK1122)/Storage (EK1100)/Term 64 (EL7332)
//     Drive/Inputs/In/nState1 @bit 3 <-> DCM Status Channel 1/Status/Error
//     Drive/Inputs/In/nState1 @bit 5 <-> DCM Status Channel 1/Status/Moving negative
//     Drive/Inputs/In/nState1 @bit 4 <-> DCM Status Channel 1/Status/Moving positive
//     Drive/Inputs/In/nState1 @bit 1 <-> DCM Status Channel 1/Status/Ready
//     Drive/Inputs/In/nState1 <-> DCM Status Channel 1/Status/Ready to enable
//     Drive/Inputs/In/nState1 @bit 6 <-> DCM Status Channel 1/Status/Torque reduced
//     Drive/Inputs/In/nState1 @bit 2 <-> DCM Status Channel 1/Status/Warning
//     Drive/Inputs/In/nState2 @bit 3 <-> DCM Status Channel 1/Status/Digital input 1
//     Drive/Inputs/In/nState2 @bit 4 <-> DCM Status Channel 1/Status/Digital input 2
//     Drive/Inputs/In/nState2 @bit 5 <-> DCM Status Channel 1/Status/Sync error
//     Drive/Inputs/In/nState2 @bit 7 <-> DCM Status Channel 1/Status/TxPDO Toggle
//     Drive/Inputs/In/nState4 @bit 1 <-> WcState/InputToggle
//     Drive/Inputs/In/nState4 <-> WcState/WcState
//     Drive/Outputs/Out/nCtrl1 <-> DCM Control Channel 1/Control/Enable
//     Drive/Outputs/Out/nCtrl1 @bit 2 <-> DCM Control Channel 1/Control/Reduce torque
//     Drive/Outputs/Out/nCtrl1 @bit 1 <-> DCM Control Channel 1/Control/Reset
//     Drive/Outputs/Out/nDataOut2[0] <-> DCM Velocity Channel 1/Velocity
//   NC-Task 1 SAF/Axes/Storage B <-> Device 3 (EtherCAT)/Term 1 (EK1100)/Storage|Casting (EK1122)/Storage (EK1100)/Term 64 (EL7332)
//     Drive/Inputs/In/nState1 @bit 3 <-> DCM Status Channel 2/Status/Error
//     Drive/Inputs/In/nState1 @bit 5 <-> DCM Status Channel 2/Status/Moving negative
//     Drive/Inputs/In/nState1 @bit 4 <-> DCM Status Channel 2/Status/Moving positive
//     Drive/Inputs/In/nState1 @bit 1 <-> DCM Status Channel 2/Status/Ready
//     Drive/Inputs/In/nState1 <-> DCM Status Channel 2/Status/Ready to enable
//     Drive/Inputs/In/nState1 @bit 6 <-> DCM Status Channel 2/Status/Torque reduced
//     Drive/Inputs/In/nState1 @bit 2 <-> DCM Status Channel 2/Status/Warning
//     Drive/Inputs/In/nState2 @bit 3 <-> DCM Status Channel 2/Status/Digital input 1
//     Drive/Inputs/In/nState2 @bit 4 <-> DCM Status Channel 2/Status/Digital input 2
//     Drive/Inputs/In/nState2 @bit 5 <-> DCM Status Channel 2/Status/Sync error
//     Drive/Inputs/In/nState2 @bit 7 <-> DCM Status Channel 2/Status/TxPDO Toggle
//     Drive/Inputs/In/nState4 @bit 1 <-> WcState/InputToggle
//     Drive/Inputs/In/nState4 <-> WcState/WcState
//     Drive/Outputs/Out/nCtrl1 <-> DCM Control Channel 2/Control/Enable
//     Drive/Outputs/Out/nCtrl1 @bit 2 <-> DCM Control Channel 2/Control/Reduce torque
//     Drive/Outputs/Out/nCtrl1 @bit 1 <-> DCM Control Channel 2/Control/Reset
//     Drive/Outputs/Out/nDataOut2[0] <-> DCM Velocity Channel 2/Velocity
//   PLC/PLC Instance <-> Device 3 (EtherCAT)/Term 1 (EK1100)/Ovens (EK1122)/Oven_A (EK1100)/Term 14 (EL1004)
//     PlcTask Inputs/MAIN._Peripherie._Handling._components.SafetyGateRef_A.LockButton.Button <-> Channel 3/MAIN._Peripherie._Handling._components.SafetyGateRef_A.LockButton.Button
//     PlcTask Inputs/MAIN._Peripherie._Handling._components.SafetyGateRef_A.RequestButton.Button <-> Channel 2/MAIN._Peripherie._Handling._components.SafetyGateRef_A.RequestButton.Button
//     PlcTask Inputs/MAIN._Peripherie._Handling._components.SafetyGateRef_A.StartButton.Button <-> Channel 1/MAIN._Peripherie._Handling._components.SafetyGateRef_A.StartButton.Button
//   PLC/PLC Instance <-> Device 3 (EtherCAT)/Term 1 (EK1100)/Ovens (EK1122)/Oven_A (EK1100)/Term 15 (EL2004)
//     PlcTask Outputs/MAIN._Peripherie._Handling._components.SafetyGateRef_A.LockButton.Light <-> Channel 3/MAIN._Peripherie._Handling._components.SafetyGateRef_A.LockButton.Light
//     PlcTask Outputs/MAIN._Peripherie._Handling._components.SafetyGateRef_A.RequestButton.Light <-> Channel 2/MAIN._Peripherie._Handling._components.SafetyGateRef_A.RequestButton.Light
//     PlcTask Outputs/MAIN._Peripherie._Handling._components.SafetyGateRef_A.StartButton.Light <-> Channel 1/MAIN._Peripherie._Handling._components.SafetyGateRef_A.StartButton.Light
//   PLC/PLC Instance <-> Device 3 (EtherCAT)/Term 1 (EK1100)/Ovens (EK1122)/Oven_B (EK1100)/Term 22 (EL1004)
//     PlcTask Inputs/MAIN._Peripherie._Handling._components.SafetyGateRef_B.LockButton.Button <-> Channel 3/MAIN._Peripherie._Handling._components.SafetyGateRef_B.LockButton.Button
//     PlcTask Inputs/MAIN._Peripherie._Handling._components.SafetyGateRef_B.RequestButton.Button <-> Channel 2/MAIN._Peripherie._Handling._components.SafetyGateRef_B.RequestButton.Button
//     PlcTask Inputs/MAIN._Peripherie._Handling._components.SafetyGateRef_B.StartButton.Button <-> Channel 1/MAIN._Peripherie._Handling._components.SafetyGateRef_B.StartButton.Button
//   PLC/PLC Instance <-> Device 3 (EtherCAT)/Term 1 (EK1100)/Ovens (EK1122)/Oven_B (EK1100)/Term 23 (EL2004)
//     PlcTask Outputs/MAIN._Peripherie._Handling._components.SafetyGateRef_B.LockButton.Light <-> Channel 3/MAIN._Peripherie._Handling._components.SafetyGateRef_B.LockButton.Light
//     PlcTask Outputs/MAIN._Peripherie._Handling._components.SafetyGateRef_B.RequestButton.Light <-> Channel 2/MAIN._Peripherie._Handling._components.SafetyGateRef_B.RequestButton.Light
//     PlcTask Outputs/MAIN._Peripherie._Handling._components.SafetyGateRef_B.StartButton.Light <-> Channel 1/MAIN._Peripherie._Handling._components.SafetyGateRef_B.StartButton.Light
//   PLC/PLC Instance <-> Device 3 (EtherCAT)/Term 1 (EK1100)/Term 33 (EL6910)
//     PlcTask Inputs/MAIN._Peripherie._Handling._components.RackFeederRef.tsAckReq <-> StandardInputs/Rackfeeder_Axis.Error_AckReq_121
//     PlcTask Inputs/MAIN._Peripherie._Handling._components.RackFeederRef.tsSS1 <-> StandardInputs/Rackfeeder_Axis.SS1_Active_82
//     PlcTask Inputs/MAIN._Peripherie._Handling._components.RackFeederRef.tsSTO <-> StandardInputs/Rackfeeder_Axis.STO_Active_84
//     PlcTask Inputs/MAIN._Peripherie._Handling._components.SafetyGateRef_A.tsOpen <-> StandardInputs/SafetyGates.Open_A_75
//     PlcTask Inputs/MAIN._Peripherie._Handling._components.SafetyGateRef_A.tsSafe <-> StandardInputs/SafetyGates.Safe_A_73
//     PlcTask Inputs/MAIN._Peripherie._Handling._components.SafetyGateRef_B.tsOpen <-> StandardInputs/SafetyGates.Open_B_76
//     PlcTask Inputs/MAIN._Peripherie._Handling._components.SafetyGateRef_B.tsSafe <-> StandardInputs/SafetyGates.Safe_B_74
//     PlcTask Inputs/MAIN._Peripherie._Handling._components.SegmentDoorRef_A.tsAckReq <-> StandardInputs/Oven_Axis.Error_AckReq_OvenA_90
//     PlcTask Inputs/MAIN._Peripherie._Handling._components.SegmentDoorRef_A.tsSS1 <-> StandardInputs/Oven_Axis.SS1_Active_OvenA_92
//     PlcTask Inputs/MAIN._Peripherie._Handling._components.SegmentDoorRef_A.tsSTO <-> StandardInputs/Oven_Axis.STO_Active_OvenA_94
//     PlcTask Inputs/MAIN._Peripherie._Handling._components.SegmentDoorRef_B.tsAckReq <-> StandardInputs/Oven_Axis.Error_AckReq_OvenB_126
//     PlcTask Inputs/MAIN._Peripherie._Handling._components.SegmentDoorRef_B.tsSS1 <-> StandardInputs/Oven_Axis.SS1_Active_OvenB_125
//     PlcTask Inputs/MAIN._Peripherie._Handling._components.SegmentDoorRef_B.tsSTO <-> StandardInputs/Oven_Axis.STO_Active_OvenB_127
//     PlcTask Inputs/MAIN._Peripherie._Handling._components.TwinSAFERef.atsEmergencyActive[0] <-> StandardInputs/TwinSafeMain.Emergency01_Active_63
//     PlcTask Inputs/MAIN._Peripherie._Handling._components.TwinSAFERef.atsEmergencyActive[1] <-> StandardInputs/TwinSafeMain.Emergency02_Active_64
//     PlcTask Inputs/MAIN._Peripherie._Handling._components.TwinSAFERef.tsComErr <-> StandardInputs/TwinSafeMain.ComErr_99
//     PlcTask Inputs/MAIN._Peripherie._Handling._components.TwinSAFERef.tsEmergencySafe <-> StandardInputs/TwinSafeMain.Safe_62
//     PlcTask Inputs/MAIN._Peripherie._Handling._components.TwinSAFERef.tsFbErr <-> StandardInputs/TwinSafeMain.FBErr_98
//     PlcTask Inputs/MAIN._Peripherie._Handling._components.TwinSAFERef.tsFbRun <-> StandardInputs/TwinSafeMain.FBRun_100
//     PlcTask Inputs/MAIN._Peripherie._Handling._components.TwinSAFERef.tsInRun <-> StandardInputs/TwinSafeMain.InRun_55
//     PlcTask Inputs/MAIN._Peripherie._Handling._components.TwinSAFERef.tsOtherErr <-> StandardInputs/TwinSafeMain.OtherErr_56
//     PlcTask Inputs/MAIN._Peripherie._Handling._components.TwinSAFERef.tsOutErr <-> StandardInputs/TwinSafeMain.OutErr_101
//     PlcTask Outputs/MAIN._Peripherie._Handling._components.RackFeederRef.tsAck <-> StandardOutputs/Rackfeeder_Axis.Error_Ack_80
//     PlcTask Outputs/MAIN._Peripherie._Handling._components.SafetyGateRef_A.tsLockCmd <-> StandardOutputs/SafetyGates.LockCmd_A_109
//     PlcTask Outputs/MAIN._Peripherie._Handling._components.SafetyGateRef_A.tsRestart <-> StandardOutputs/SafetyGates.Restart_A_71
//     PlcTask Outputs/MAIN._Peripherie._Handling._components.SafetyGateRef_B.tsLockCmd <-> StandardOutputs/SafetyGates.LockCmd_B_110
//     PlcTask Outputs/MAIN._Peripherie._Handling._components.SafetyGateRef_B.tsRestart <-> StandardOutputs/SafetyGates.Restart_B_72
//     PlcTask Outputs/MAIN._Peripherie._Handling._components.SegmentDoorRef_A.tsAck <-> StandardOutputs/Oven_Axis.Error_Ack_OvenA_122
//     PlcTask Outputs/MAIN._Peripherie._Handling._components.SegmentDoorRef_B.tsAck <-> StandardOutputs/Oven_Axis.Error_Ack_OvenB_88
//     PlcTask Outputs/MAIN._Peripherie._Handling._components.TwinSAFERef.tsDriveRestart <-> StandardOutputs/TwinSafeMain.DriveRestart_117
//     PlcTask Outputs/MAIN._Peripherie._Handling._components.TwinSAFERef.tsEmergencyRestart <-> StandardOutputs/TwinSafeMain.Restart_61
//     PlcTask Outputs/MAIN._Peripherie._Handling._components.TwinSAFERef.tsErrAck <-> StandardOutputs/TwinSafeMain.ErrAck_53
//     PlcTask Outputs/MAIN._Peripherie._Handling._components.TwinSAFERef.tsRunStop <-> StandardOutputs/TwinSafeMain.RunStop_54
//   PLC/PLC Instance <-> NC-Task 1 SAF/Axes/Oven A
//     PlcTask Inputs/MAIN._Peripherie._Handling._components.SegmentDoorRef_A.VertikalAxis.NcToPlc <-> Outputs/ToPlc
//     PlcTask Outputs/MAIN._Peripherie._Handling._components.SegmentDoorRef_A.VertikalAxis.PlcToNc <-> Inputs/FromPlc
//   PLC/PLC Instance <-> NC-Task 1 SAF/Axes/Oven A CH1
//     PlcTask Inputs/MAIN._Peripherie._Handling._components.SegmentDoorRef_A.LatchLeft.NcToPlc <-> Outputs/ToPlc
//     PlcTask Outputs/MAIN._Peripherie._Handling._components.SegmentDoorRef_A.LatchLeft.PlcToNc <-> Inputs/FromPlc
//   PLC/PLC Instance <-> NC-Task 1 SAF/Axes/Oven A CH2
//     PlcTask Inputs/MAIN._Peripherie._Handling._components.SegmentDoorRef_A.LatchRight.NcToPlc <-> Outputs/ToPlc
//     PlcTask Outputs/MAIN._Peripherie._Handling._components.SegmentDoorRef_A.LatchRight.PlcToNc <-> Inputs/FromPlc
//   PLC/PLC Instance <-> NC-Task 1 SAF/Axes/Oven B
//     PlcTask Inputs/MAIN._Peripherie._Handling._components.SegmentDoorRef_B.VertikalAxis.NcToPlc <-> Outputs/ToPlc
//     PlcTask Outputs/MAIN._Peripherie._Handling._components.SegmentDoorRef_B.VertikalAxis.PlcToNc <-> Inputs/FromPlc
//   PLC/PLC Instance <-> NC-Task 1 SAF/Axes/Oven B CH1
//     PlcTask Inputs/MAIN._Peripherie._Handling._components.SegmentDoorRef_B.LatchLeft.NcToPlc <-> Outputs/ToPlc
//     PlcTask Outputs/MAIN._Peripherie._Handling._components.SegmentDoorRef_B.LatchLeft.PlcToNc <-> Inputs/FromPlc
//   PLC/PLC Instance <-> NC-Task 1 SAF/Axes/Oven B CH2
//     PlcTask Inputs/MAIN._Peripherie._Handling._components.SegmentDoorRef_B.LatchRight.NcToPlc <-> Outputs/ToPlc
//     PlcTask Outputs/MAIN._Peripherie._Handling._components.SegmentDoorRef_B.LatchRight.PlcToNc <-> Inputs/FromPlc
//   PLC/PLC Instance <-> NC-Task 1 SAF/Axes/Rackfeeder Teleskop
//     PlcTask Inputs/MAIN._Peripherie._Handling._components.RackFeederRef.TelescopeAxis.NcToPlc <-> Outputs/ToPlc
//     PlcTask Outputs/MAIN._Peripherie._Handling._components.RackFeederRef.TelescopeAxis.PlcToNc <-> Inputs/FromPlc
//   PLC/PLC Instance <-> NC-Task 1 SAF/Axes/Rackfeeder X
//     PlcTask Inputs/MAIN._Peripherie._Handling._components.RackFeederRef.HorizontalAxis.NcToPlc <-> Outputs/ToPlc
//     PlcTask Outputs/MAIN._Peripherie._Handling._components.RackFeederRef.HorizontalAxis.PlcToNc <-> Inputs/FromPlc
//   PLC/PLC Instance <-> NC-Task 1 SAF/Axes/Rackfeeder Y
//     PlcTask Inputs/MAIN._Peripherie._Handling._components.RackFeederRef.VerticalAxis.NcToPlc <-> Outputs/ToPlc
//     PlcTask Outputs/MAIN._Peripherie._Handling._components.RackFeederRef.VerticalAxis.PlcToNc <-> Inputs/FromPlc

CONFIGURATION PLC
    RESOURCE PLC ON TwinCAT3
        TASK PlcTask(INTERVAL := T#10ms, PRIORITY := 20);
        PROGRAM MAIN WITH PlcTask : MAIN;
    END_RESOURCE
END_CONFIGURATION

// ---- Components/ST_MachineSetting.TcDUT
TYPE ST_MachineSetting :
STRUCT
//	astWorkpiecePlaceStates					: ARRAY[0..GVL.nMaxWorkpiecePlaceStatus] OF TcaWorkpiecePlaceStatus;
//	astWorkpieceType						: ARRAY[0..GVL.nMaxWorkpieceTyp] OF ST_WorkpieceType;
END_STRUCT
END_TYPE

// ---- Components/TcaCarrier/Structures/TcaCarrierConfig.TcDUT
TYPE TcaCarrierConfig :
STRUCT	
	/// Geometry
	Layout : eTcaCarrierLayout;		
	PositionsInRow : INT;			// Numbers of Positions in first Row
	RowDistance : REAL;		// Distance from one Row to the other
	PositionsInColumn : INT;			// Numbers of Positions in one Column
	ColumnDistance : REAL;		// Distance from one Column to the other
	CoordinateFirstWorkpiece : ST_Coordinate;
	
	InitialStatus : eTcaWorkpiecePlaceStatus;
	RequestStatus : eTcaWorkpiecePlaceStatus;	
	

END_STRUCT
END_TYPE

// ---- Components/TcaCarrier/Structures/TcaCarrierService.TcDUT
TYPE TcaCarrierService :
STRUCT
	WorkpiecePlaces : INT; // starts with 1
	PrimaryWorkpieceStatusCount : INT;
	SecondaryWorkpieceStatusCount : INT;
	PrimaryWorkpieceStatusColor : COLOR;
	SecondaryWorkpieceStatusColor : COLOR;
	ConfigError	: BOOL;
END_STRUCT
END_TYPE

// ---- Components/TcaCarrier/Structures/TcaCarrierData.TcDUT
TYPE TcaCarrierData :
STRUCT	
	Enabled : BOOL;
	Id : INT;
	Logging : WSTRING;	// Information in csv, xml or json Format
	Error : BOOL;	

	/// Geometry
	//eConfiguration : eTcaCarrierConfig;		
	//PositionsInRow : INT;			// Numbers of Positions in first Row
	//RowDistance : REAL;		// Distance from one Row to the other
	//PositionsInColumn : INT;			// Numbers of Positions in one Column
	//ColumnDistance : REAL;		// Distance from one Column to the other
	//CoordinateFirstWorkpiece : ST_Coordinate;
	//CoordinateLastWorkpiece : ST_Coordinate;
	
	InitialStatus : eTcaWorkpiecePlaceStatus;
	RequestStatus : eTcaWorkpiecePlaceStatus;	

	WorkpiecesEnabled : ARRAY[0..TcaCarrier.MAX_WORKPIECEPLACES] OF BOOL;
	WorkpiecesCoordinate : ARRAY[0..TcaCarrier.MAX_WORKPIECEPLACES] OF ST_Coordinate;
	WorkpiecesData : ARRAY[0..TcaCarrier.MAX_WORKPIECEPLACES] OF TcaWorkpiecePlaceData;
	

END_STRUCT
END_TYPE

// ---- Components/TcaPushButton/Enumerations/eTcaPushButtonColor.TcDUT
{attribute 'qualified_only'}
{attribute 'strict'}
TYPE eTcaPushButtonColor :
(
	none := 0,
	Green := 1,
	Red := 2,
	Yellow := 3,
	Blue := 4,
	Orange := 5,
	custom := 6,
	white := 7
);
END_TYPE

// ---- Components/TcaPushButton/Enumerations/eTcaPushButtonLightState.TcDUT
{attribute 'qualified_only'}
{attribute 'strict'}
TYPE eTcaPushButtonLightState :
(
	none := 0,
	permanent := 1,
	intervall := 2
);
END_TYPE

// ---- Components/TcaPushButton/Structures/TcaPushButtonService.TcDUT
TYPE TcaPushButtonService :
STRUCT
	Button : BOOL;
	Light : BOOL;	
END_STRUCT
END_TYPE

// ---- Components/TcaStorage/eTcaStorageCmd.TcDUT
{attribute 'qualified_only'}
{attribute 'strict'}
{attribute 'to_string'}
TYPE eTcaStorageCmd :
(
	noCmd := 0,
	FillCarrier,
	RemoveCarrier,
	EmptyCarrier
);
END_TYPE

// ---- Components/TcaStorage/TcaStorageRef.TcDUT
TYPE TcaStorageRef :
STRUCT
	Sensor AT%I* : BOOL;	
END_STRUCT
END_TYPE

// ---- Components/TcaTrolley/Structures/TcaTrolleyData.TcDUT
TYPE TcaTrolleyData : 
STRUCT
	Enabled : BOOL;
	Id : INT;
	Logging : WSTRING;	// Information in csv, xml or json Format
	Error : BOOL;
	
	/// Geometry
	NumberOfCarriers : INT;	// Numbers of Positions in first Row
	CoordinateFirstCarrier : ST_Coordinate;
	CoordinateLastCarrier : ST_Coordinate;
		
	InitialStatus : eTcaWorkpiecePlaceStatus;
	RequestStatus : eTcaWorkpiecePlaceStatus;	
		
	CarrierData : ARRAY[0..TcaTrolley.MAX_CARRIERPLACES] OF TcaCarrierData;
	
END_STRUCT
END_TYPE

// ---- Components/TcaTrolley/Structures/TcaTrolleyService.TcDUT
TYPE TcaTrolleyService :
STRUCT

END_STRUCT
END_TYPE

// ---- Components/TcaTrolley_old/CMD_Trolley.TcDUT
TYPE CMD_Trolley :
STRUCT
	cmd			: eTcaTrolleyCmd;
	nId			: INT;
END_STRUCT
END_TYPE

// ---- Components/TcaWorkpiecePlace/Enumerations/eTcaWorkpiecePlaceStatus.TcDUT
{attribute 'qualified_only'}
{attribute 'strict'}
{attribute 'to_string'}
TYPE eTcaWorkpiecePlaceStatus :
(
	undefined := 0,
	noProcessDone,
	laserProcessDone,
	bondingAgentProcessDone,
	castingProcessDone,
	finishProcessDone,
	
	MAXSIZE
);
END_TYPE

// ---- Components/TcaWorkpiecePlace/Enumerations/eTcaWorkpiecePlaceShape.TcDUT
{attribute 'qualified_only'}
{attribute 'strict'}
{attribute 'to_string'}
TYPE eTcaWorkpiecePlaceShape :
(
	undefined := 0,
	roll,
	ring,
	plate,
	other,
	
	MAXSIZE
);
END_TYPE

// ---- Components/TcaWorkpiecePlace/Structures/TcaWorkpiecePlaceService.TcDUT
TYPE TcaWorkpiecePlaceService :
STRUCT

END_STRUCT
END_TYPE

// ---- Components/TcaWorkpiecePlace/Structures/TcaWorkpiecePlaceData.TcDUT
TYPE TcaWorkpiecePlaceData : 
STRUCT
	Enabled : BOOL; // tot wird nicht mehr benötigt
	Id : INT;	// <> 0 Workpiece Present 
	Error : BOOL;
	SerialNumber : STRING;
	CurrentStatus : eTcaWorkpiecePlaceStatus;
	RequestStatus : eTcaWorkpiecePlaceStatus;
	Shape : eTcaWorkpiecePlaceShape;
	Volume : ST_Coordinate;
	Logging : WSTRING;	// Information in csv, xml or json Format
	
	
END_STRUCT
END_TYPE

// ---- Components_RMTH/TcaEngelCasting/TcaEngelCastingCarrierJobStatus.TcDUT
TYPE TcaEngelCastingCarrierJobStatus :
STRUCT
	CarrierPresent : BOOL;						// TRUE wenn ein Werkstückträger abgelegt wurde
	Carrier : TcaEngelCastingCarrierStatus;		// Status des Carriers der abgelegt wurde
	Done : BOOL;								// Job wurde erfolgreich ausgeführt
	Busy : BOOL;								// Job wird ausgeführt
	Error : BOOL;								// Job endet mit Fehler
	ErrorID : INT;								// TODO: Welche unterschiedlichen Fehler sollen berücksichtigt werden? z.b: kein Blech, Ofentür offen, Wagen ist zum wechseln, ...								
END_STRUCT
END_TYPE

// ---- Components_RMTH/TcaLaserDistanceSenor/Structures/TcaLaserDistanceSenorStatus.TcDUT
TYPE
    TcaLaserDistanceSenorStatus :
    STRUCT
		{attribute addProperty Name "<#Raw range#>"}
        RawRange : REAL;
		{attribute addProperty Name "<#Real range#>"}
        RealRange : REAL;
		{attribute addProperty Name "<#Scaled value#>"}
        Scaled : REAL;
    END_STRUCT
END_TYPE

// ---- Components_RMTH/TcaRackFeeder/Structures/TcaRackFeederStatus.TcDUT
TYPE TcaRackFeederStatus :
STRUCT
    ActionDescription : STRING(100);	         
	Safe : BOOL;
END_STRUCT
END_TYPE

// ---- Components_RMTH/TcaSafetyGate/Structures/TcaSafetyGateRef.TcDUT
TYPE TcaSafetyGateRef :
STRUCT
	// Components
	StartButton	: TcaPushButtonRef;
	RequestButton : TcaPushButtonRef;	
	LockButton : TcaPushButtonRef;
	
	// SafetyPorts                    
	tsSafe AT%I* : BOOL;
	tsOpen AT%I* : BOOL;
	tsRestart AT%Q* : BOOL;    
	tsLockCmd AT%Q* : BOOL;
	
END_STRUCT
END_TYPE

// ---- Components_RMTH/TcaSafetyGate/Structures/TcaSafetyGateService.TcDUT
TYPE TcaSafetyGateService :
STRUCT
	StartButton : TcaPushButtonService;
	RequestButton : TcaPushButtonService;
	LockButton : TcaPushButtonService;
	
	Safe : BOOL;
	Open : BOOL;
	ComponentsAreService : BOOL;
END_STRUCT
END_TYPE

// ---- Components_RMTH/TcaSafetyGate/Structures/TcaSafetyGateStatus.TcDUT
TYPE TcaSafetyGateStatus :
STRUCT
    ActionDescription : STRING(100);	         
	Safe : BOOL;
	Open : BOOL;
	ComponentsAreService : BOOL;
	
END_STRUCT
END_TYPE

// ---- Components_RMTH/TcaTwinSAFE/Structures/TcaTwinSAFEConfig.TcDUT
TYPE TcaTwinSAFEConfig :
STRUCT
END_STRUCT
END_TYPE

// ---- Items/COLOR.TcDUT
TYPE COLOR : ARRAY[0..3] OF LREAL; END_TYPE

// ---- Items/ST_ComboboxEntry.TcDUT
TYPE ST_ComboboxEntry :
STRUCT    
	id : INT;
    text : STRING;
    value : INT;
END_STRUCT
END_TYPE

// ---- Items/ST_WorkpieceType.TcDUT
TYPE ST_WorkpieceType EXTENDS ST_ComboboxEntry:
STRUCT
	aColor				: COLOR;
END_STRUCT
END_TYPE

// ---- Template/Component_Cylinder/Structs/CylinderConfig.TcDUT
TYPE CylinderConfig :
STRUCT
	TimeToReachHomePosition : TIME := T#10S;
	TimeToReachWorkPosition : TIME := T#10S;
END_STRUCT
END_TYPE

// ---- Template/Component_Cylinder/Structs/TcoCylinderConfig.TcDUT
TYPE TcoCylinderConfig :
STRUCT
	TimeToReachHomePosition : TIME := T#10S;
	TimeToReachWorkPosition : TIME := T#10S;
	TimeToRefill : TIME := T#1000MS;
END_STRUCT
END_TYPE

// ---- Template/Component_Cylinder/Structs/TcoCylinderStatus.TcDUT
TYPE TcoCylinderStatus :
STRUCT
	ActionDescription : STRING(100);	
END_STRUCT
END_TYPE

// ---- Template/RackFeeder/CMD_RackFeeder.TcDUT
TYPE CMD_RackFeeder :
STRUCT
	cmd			: E_RackFeederCmd;
	nId			: INT;
END_STRUCT
END_TYPE

// ---- Template/RackFeeder/Structure/ST_RackFeederIO.TcDUT
TYPE ST_RackFeederIO :
STRUCT	
	ioAxisTraverse					: ST_AxisIO;
	ioAxisLift						: ST_AxisIO;
	ioAxisTelescope					: ST_AxisIO;	
	
	ioCarrierPresent				: ST_DigitalInputIO;
	
END_STRUCT
END_TYPE

// ---- Template/Component_Carousell/Structs/eTcoCarouselDirection.TcDUT
TYPE eTcoCarouselDirection :
(
	Cw := 0,
	Ccw := 1
);
END_TYPE

// ---- Template/Component_Carousell/Structs/TcoCarouselConfig.TcDUT
(*~
<docu>
	<summary>
		`TcoCarousel` settings/config structure.								
	</summary>				
</docu>	
~*)
TYPE
    TcoCarouselConfig :
    STRUCT

        Direction   : eTcoCarouselDirection;
  		InfoTime : TIME := T#2S;
        ErrorTime : TIME := T#5S;
		NumberOfPositions:UINT;
		// Offset in respect to frist position.
		Offset : UINT;
   
		
    END_STRUCT
END_TYPE

// ---- Template/Component_Carousell/Structs/TcoCarouselStatus.TcDUT
(*~
<docu>
	<summary>
		`TcCarousel` status structure.								
	</summary>				
</docu>	
~*)
TYPE
    TcoCarouselStatus :
    STRUCT
      	ActionDescription : STRING(100);	
        {attribute addProperty Name "<#In position#>"}
        InPosition : BOOL;
        {attribute addProperty Name "<#In precise position#>"}
        InPrecisePosition : BOOL;
        {attribute addProperty Name "<#Turn safety condition#>"}
        TurnSafetyCondition : BOOL;
        {attribute addProperty Name "<#Current position#>"}
		CurrentPosition : UINT;
        {attribute addProperty Name "<#Expected next position#>"}
		ExpectedNextPosition : UINT;
		{attribute addProperty Name "<#Positions#>" }
		Positions : ARRAY[0..20] OF UINT;

	
		
		
    END_STRUCT
END_TYPE

// ---- Utilities/Component/Enumerations/E_ComponentState.TcDUT
{attribute 'qualified_only'}
{attribute 'strict'}
TYPE E_ComponentState :
(
	none := 0,				/// Component state not set
	resetting := 1,			/// Component is resetting
	ready := 2,				/// Component is ready
	running := 3,			/// Component is running
	stopped := 4,			/// Component stopped
	error := 5				/// Component has error
);
END_TYPE

// ---- Utilities/Component/Structures/ST_ComponentVisu.TcDUT
TYPE ST_ComponentVisu :
STRUCT
	sName				: STRING;
	bError				: BOOL;
	bRunning			: BOOL;
	bReset				: BOOL;
	bEnable				: BOOL;
	bAccessPermit		: BOOL;
	eState				: E_ComponentState;
	colBackground		: DWORD;
END_STRUCT
END_TYPE

// ---- Utilities/EventLog/Enumerations/E_LoggingProvider.TcDUT
TYPE E_LoggingProvider :
(
	///kein Loggingprovider
	eLoggingProviderNone := 0,
	///Filesystem-Loggingprovider
	eLoggingProviderFile := 1,
	///Datenbank-Loggingprovider
	eLoggingProviderDataBase := 2,
	///EventLog-Loggingprovider
	eLoggingProviderEventLog := 3,
	eLoggingProviderNetSvc := 4
);
END_TYPE

// ---- Utilities/EventLog/Enumerations/E_Priority.TcDUT
/// enumeration of all possible priority
TYPE E_Priority :
(
	/// no priority
	ePriority_none := 0,
	/// info priority
	ePriority_info := 1,
	/// warn priority
	ePriority_warning := 2,
	/// error priority -> Zyklusstop
	ePriority_fault := 3,
	/// error priority with fast stop -> Stopp im aktuellen Schritt 
	ePriority_faultFastStop := 4,
	/// error priority with emergency stop -> Sofortstop aller Objekte
	ePriority_faultEmergency := 5
);
END_TYPE

// ---- Utilities/EventLog/E_Event.TcDUT
/// enumeration of all possible notifications
TYPE E_Event :
(
	/// notification not set
	eEvent_none := 0,
	
	eEvent_generalError := 1,
	eEvent_generalWarning := 2,
	eEvent_generalInfo := 3,
	
	/// - code errors -
	/// code error (e.g.: check bounds, check div, ...) -> additional info (error details/index/location) in dynamic content var
	eEvent_codeError := 11,
	/// - system errors -
	/// system error (e.g.: (re)started, cycletime exceeded, ...) -> additional info (index/location) in dynamic content var
	eEvent_systemError := 12,
	/// - HW errors -
	/// hardware error -> additional info (error details/index/location) in dynamic content var
	eEvent_hardwareError := 13,
	/// hardware warning -> additional info (error details/index/location) in dynamic content var
	eEvent_hardwareWarning := 14,
	/// EtherCAT Master Fehler
	eEvent_EcMasterError := 15,
	/// EtherCAT Slave Fehler
	eEvent_EcSlaveError := 16,
    
	// - Safety system errors -
	/// safety error -> additional info (error details/index/location) in dynamic content var
	eEvent_safetyError := 17,
	
	// - Unit Test Meldungen
	v_unitTest := 18,
	
	// bis 09
	
	// Cabinet errors
	/// Feld01 - xxx
	eEvent_Cabinet01 := 100,
	/// Feld02 - xxx
	eEvent_Cabinet02 := 110,
	/// Feld03 - xxx
	eEvent_Cabinet03 := 120,
	
	
	
	// bis 40
	
	// 40 -> Transfer System
	eEvent_transferSystemError := 40,
	
	// 50 -> Safety Fehler Schutztüre, Not-Halt, ...
	eEvent_safetyNotHalt := 50,
	eEvent_safetyArea_Machine := 51,
	eEvent_safetyArea_Robo1 := 52,
	eEvent_safetyArea_SAA := 53,
	eEvent_safetyArea_Robo2 := 54,
	eEvent_safetyArea_PA := 55

);
END_TYPE

// ---- Utilities/EventLog/Structures/ST_EventBase.TcDUT
/// Event structure
TYPE ST_EventBase :
STRUCT
	eMachineArea		: E_MachineArea;
	eComponent			: E_ComponentType;
	nComponentID		: INT;
	refComponent		: REFERENCE TO FB_Component;
	
	eEventID			: E_Event;
	
	ePriority			: E_Priority;
	bSignalize			: BOOL;
	
	sPosition			: T_MaxString;
	sDescription		: T_MaxString;
END_STRUCT
END_TYPE

// ---- Utilities/EventLog/Structures/ST_EventVisu.TcDUT
/// Event structure
TYPE ST_EventVisu :
STRUCT
	ucTable				: Uc_EventLogTable;
	ucControl			: Uc_EventLogControl;
	
END_STRUCT
END_TYPE

// ---- Utilities/Helpers/Color/ST_ColorCMYK.TcDUT
TYPE ST_ColorCMYK :
STRUCT
	nCyan						: BYTE;
	nMagenta					: BYTE;
	nYellow						: BYTE;
	nKey						: BYTE;
END_STRUCT
END_TYPE

// ---- Utilities/Helpers/E_OperationResult.TcDUT
{attribute 'qualified_only'}
{attribute 'strict'}
TYPE E_OperationResult :
(
	None := 0,		/// operation result not initialized
	Busy,			/// operation process busy
	Ok,				/// operation succeeded or true
	NOk,			/// operation result not ok or false
	Error			/// operation failed/error
);
END_TYPE

// ---- Utilities/Helpers/ST_DefaultPulse.TcDUT
TYPE ST_DefaultPulse :
STRUCT
	/// default impulse flags
	bImpulse1000ms: BOOL;
	bImpulse500ms: BOOL;
	bImpulse300ms: BOOL;
	bImpulse200ms: BOOL;
	bImpulse100ms: BOOL;
	/// default toggle flags
	bToggle1000ms: BOOL;
	bToggle500ms: BOOL;
	bToggle300ms: BOOL;
	bToggle200ms: BOOL;
	bToggle100ms: BOOL;
END_STRUCT
END_TYPE

// ---- Utilities/Helpers/ST_PlcSystemInfo.TcDUT
TYPE ST_PlcSystemInfo :
STRUCT
	/// system info structure
	stPlcAppSystemInfo: PlcAppSystemInfo;
	/// tast info structure
	stPlcTaskSystemInfo: PlcTaskSystemInfo;
	/// cycle time from task configuration in [s]
	fCycleTime: LREAL;
	/// needed cycletime for the last cycle in [s]
	fLastExecTime: LREAL;
END_STRUCT
END_TYPE

// ---- Utilities/List/Structures/ST_Listentry.TcDUT
TYPE ST_Listentry :
STRUCT
	nRawId		: INT;
	nId			: INT;
	bEnable		: BOOL;
	sName		: STRING;
END_STRUCT
END_TYPE

// ---- Utilities/StaticsConstant.TcGVL
VAR_GLOBAL CONSTANT
	sEmpty: STRING(0) := '';
	dtMinValue: DT := DATE_AND_TIME#1970-1-1-0:0;
	dtMaxValue: DT := DATE_AND_TIME#2106-2-6-6:28:15;
	iLogArraySize: INT := 500;
END_VAR

// ---- Components/TcaCarrier/ITcaCarrier.TcIO
INTERFACE ITcaCarrier

METHOD ChangeData : ITcoTaskStatus 
VAR_INPUT
	inData : TcaCarrierData;
END_VAR
END_METHOD

METHOD CoordinatesOf : ST_Coordinate
VAR_INPUT
	WorkpiecePlace		: INT;
END_VAR
END_METHOD

METHOD CountEmptyPlaces : INT
END_METHOD

METHOD CountPlacesByStatus : INT
VAR_INPUT
	nStatus			: INT;
END_VAR
END_METHOD

METHOD FillWithWorkpieces_CustomStatus : ITcoTaskStatus
VAR_INPUT
	Status		: eTcaWorkpiecePlaceStatus;
END_VAR
END_METHOD

METHOD FillWithWorkpieces_InitialStatus : ITcoTaskStatus
VAR_INPUT
END_VAR
END_METHOD

METHOD FillWithWorkpieces_RequestStatus : ITcoTaskStatus
VAR_INPUT
END_VAR
END_METHOD

METHOD FindPlace : REFERENCE TO TcaWorkpiecePlace //-1..no Position found

VAR_INPUT
	Status		: eTcaWorkpiecePlaceStatus;
END_VAR
END_METHOD

METHOD GetPlaceReference : REFERENCE TO TcaWorkpiecePlace
VAR_INPUT
	nIndexNr		: INT;
END_VAR
END_METHOD

METHOD RefreshStatus : BOOL
END_METHOD

END_INTERFACE

// ---- Utilities/EventLog/Interface/ITFLoggingProvider.TcIO
INTERFACE ITFLoggingProvider

/// Add log method
{attribute 'object_name' := 'AddLog'}
METHOD AddLog : BOOL
VAR_INPUT
	/// log message 
	sText: T_MaxString;
	/// log source
	sSource: STRING;
	///	level: eLogLevelNone, eLogLevelError, eLogLevelWarning, eLogLevelInformation	
	eLevel: E_LogLevel;
END_VAR
END_METHOD

{attribute 'object_name' := 'Run'}
METHOD Run
END_METHOD

END_INTERFACE

// ---- Program/MAIN.TcPOU
PROGRAM MAIN
VAR
	_Peripherie	: Peripherie;
	
END_VAR

_Peripherie.Run();
_Peripherie.RtcSynchronize(TRUE, '', 60);

END_PROGRAM

// ---- Program/Peripherie.TcPOU
FUNCTION_BLOCK Peripherie EXTENDS TcoCore.TcoContext
VAR
	_Handling : Handling(THIS^);
	
	_Trolley : TcaTrolley(THIS^);
	
	_Carrier : TcaCarrier(THIS^);
END_VAR

VAR
	apply				: BOOL;
END_VAR

(*~
	<docu>
		<summary>
			Main method of the TcoContext. This is the entry point of any control logic that belongs to this context. 
			The call of this method is ensured by calling the <c>InstanceName.Run()</c> method, and it must not be called explicitly.
			This method is abstract, and it must be overridden in derived block.
		</summary>
	</docu>
~*)
METHOD PROTECTED  Main
THIS^.RtcSynchronize(TRUE, '', 60);
_Handling();

IF apply THEN
	apply := FALSE;
	_Carrier.ApplyConfig();
END_IF
END_METHOD

END_FUNCTION_BLOCK

// ---- Program/Handling/Handling.TcPOU
FUNCTION_BLOCK Handling EXTENDS TcoCore.TcoObject 
VAR
	_components : Handling_Components(THIS^);	
	
	_WorkpiecePlace : TcaWorkpiecePlace(THIS^);
	_Carrier : TcaCarrier(THIS^);
	_Storage : TcaStorage(THIS^);

	_groundMode : Handling_GroundMode(THIS^, eRestoreMode.None);
	_openDoor : Handling_OpenDoor(THIS^, eRestoreMode.None);
	
	_groundModeTask : TcoCore.TcoTask(THIS^);
	_openDoorTask : TcoCore.TcoTask(THIS^);
	

	_enable1			: BOOL := TRUE;
	_enablePositive1    : BOOL := TRUE;
	_enableNegative1    : BOOL := TRUE;
	_calibrationCam1    : BOOL := TRUE;
	
END_VAR

_components();




//_Storage();
//_Storage.Service();
//
//_Carrier();
//_Carrier.Service();
//
//_WorkpiecePlace();
//_WorkpiecePlace.Service();

// open Door Task
_openDoorTask.Enabled := _groundModeTask.Done;
IF(_openDoorTask.Execute()) THEN
	Messenger.Trace('Openb Door active');
	
	_openDoor.Run();
	_openDoorTask.DoneWhen(_openDoor.CurrentStep.ID = 300);
	IF _openDoorTask.Done THEN
		_openDoorTask.Restore();	
		_openDoor.Restore();
	END_IF	
END_IF


// ground Mode Task
IF(_groundModeTask.Execute()) THEN
	Messenger.Trace('Ground position mode active');
	_openDoorTask.Restore();
	_openDoor.Restore();
	
	_groundMode.Run();
	_groundModeTask.DoneWhen(_groundMode.CurrentStep.ID = 300);
	IF _groundModeTask.Done THEN
		_groundMode.Restore();
	END_IF
END_IF

PROPERTY Components : REFERENCE TO Handling_Components
GET
Components REF= _components;
END_GET
END_PROPERTY

END_FUNCTION_BLOCK

// ---- Components/TcaWorkpiecePlace/TcaWorkpiecePlace.TcPOU
FUNCTION_BLOCK TcaWorkpiecePlace EXTENDS TcoCore.TcoComponent

VAR CONSTANT
	MAX_PROGRESSSTEPS : INT := 127;
END_VAR

VAR PERSISTENT
    _carrier : ITcaCarrier;	
	_data : TcaWorkpiecePlaceData;
	//_config : TcaWorkpiecePlaceConfig;
	//_service : TcaWorkpiecePlaceService;
END_VAR

VAR
	_onCarrier : BOOL;
	_modifyTask	: TcoCore.TcoTask(THIS^);
END_VAR

IF _modifyTask.Execute() THEN
	
	IF Carrier <> 0 THEN
		Carrier.RefreshStatus();
	END_IF
	
	_modifyTask.DoneWhen(TRUE);
END_IF

IF _modifyTask.Done THEN
	_modifyTask.Restore();
END_IF

PROPERTY Carrier : ITcaCarrier
GET
VAR
	tmpPointer 	: POINTER TO TcaCarrier;
END_VAR
IF _onCarrier THEN 
	Carrier := _carrier;  
END_IF
END_GET
END_PROPERTY

PROPERTY Data : REFERENCE TO TcaWorkpiecePlaceData
GET
Data REF= _data;
END_GET
SET
_data := Data;
END_SET
END_PROPERTY

PROPERTY Enabled : BOOL
GET
Enabled := _data.Enabled;
END_GET
SET
_data.Enabled := Enabled;
END_SET
END_PROPERTY

PROPERTY Error : BOOL
GET
Error := _data.Error;
END_GET
SET
_data.Error := Error;
END_SET
END_PROPERTY

{attribute 'hide'}
METHOD FB_init : BOOL
VAR_INPUT
	bInitRetains : BOOL; // if TRUE, the retain variables are initialized (warm start / cold start)
	bInCopyCode : BOOL;  // if TRUE, the instance afterwards gets moved into the copy code (online change)
	ParentObject : ITcoObject;
END_VAR
IF __QUERYINTERFACE(_ParentObject,_carrier) THEN 	// Check if _Parent is Carrier
	_onCarrier := TRUE;
ELSE
	_onCarrier := FALSE;
END_IF
END_METHOD

PROPERTY Id : INT
GET
Id := _data.Id;
END_GET
SET
_data.Id := Id;
END_SET
END_PROPERTY

PROPERTY ModifyTask : TcoCore.ITcoTask
GET
ModifyTask := _modifyTask;
END_GET
END_PROPERTY

(*~
	<docu>
		<summary>
			Restores this instance to the Ready state. Can be called explicitly or from within one of the restore mechanisms.	
		</summary>			
	</docu>	
~*)
METHOD  Restore : ITcoRestorable
_data.Error := FALSE;
_data.SerialNumber := '';
_data.Logging := "";
END_METHOD

(*~
	<docu>
		<summary>
		    Custom service (manual, maintenance) logic.
			This method must be implemented in derived class.
		</summary>			
	</docu>	
~*)
METHOD PROTECTED  ServiceMode
END_METHOD

PROPERTY WorkpiecePresent : BOOL
GET
WorkpiecePresent := _data.Id <> 0;
END_GET
END_PROPERTY

END_FUNCTION_BLOCK

// ---- Components/TcaCarrier/TcaCarrier.TcPOU
FUNCTION_BLOCK TcaCarrier EXTENDS TcoCore.TcoComponent IMPLEMENTS ITcaCarrier
VAR CONSTANT
	MAX_WORKPIECEPLACES : INT := 127;
END_VAR

VAR PERSISTENT
	_carrierID : INT;	
	_data : TcaCarrierData;
	_config : TcaCarrierConfig;
	_arrayOfWorkpiecePlaces : ARRAY[0..MAX_WORKPIECEPLACES] OF TcaWorkpiecePlace(THIS^);
END_VAR

VAR
	_ModifyTask : TcaCarrierModifyTask(THIS^);	
	_modifyId : INT := 0;
	_i : INT;
		
	_WorkpieceStatusCount : ARRAY[0..eTcaWorkpiecePlaceStatus.MAXSIZE] OF INT;
	_PrimaryStatus : eTcaWorkpiecePlaceStatus;
	_SecondaryStatus : eTcaWorkpiecePlaceStatus;
	_PrimaryStatusCount : INT;
	_SecondaryStatusCount : INT;
	
	_ConfigError	: BOOL;
	
END_VAR

THIS^._ModifyTask(inoArrayOfWorkpiecePlaces := _arrayOfWorkpiecePlaces);

FOR _i:= 0 TO MAX_WORKPIECEPLACES DO
	_arrayOfWorkpiecePlaces[_i]();
END_FOR

METHOD ApplyConfig : REFERENCE TO TcaCarrier
VAR
	tmpData				: TcaCarrierConfig;
	
	tmpOffset 			: REAL;
	tmpOddRow			: INT;
	tmpEvenRow			: INT;
	tmpWorkpieceCount	: INT;
	
	tmpPos		 		: INT;
	tmpLoc		 		: INT;		
	tmpRow 				: INT;
	//tmpLvl				: INT;
	
	nRowNumber			: INT;
	nLocationNumber		: INT; 
	
	ni					: INT;
	
	tmpCoordinate 		: ST_Coordinate;		
END_VAR
tmpData := _config;

CASE tmpData.Layout OF
	eTcaCarrierLayout.Layout1 : 
		tmpOffset := 0;
		tmpOddRow := tmpData.PositionsInRow;
        tmpEvenRow := tmpData.PositionsInRow;
        tmpWorkpieceCount := tmpData.PositionsInRow*tmpData.PositionsInColumn;
		
    eTcaCarrierLayout.Layout2 :
		tmpOffset := 0.5;
		tmpOddRow := tmpData.PositionsInRow;
		tmpEvenRow := tmpData.PositionsInRow;
        tmpWorkpieceCount := tmpData.PositionsInRow*tmpData.PositionsInColumn;
		 
    eTcaCarrierLayout.Layout3 :
		 tmpOffset := -0.5;
		 tmpOddRow := tmpData.PositionsInRow;
         tmpEvenRow := tmpData.PositionsInRow;
         tmpWorkpieceCount := tmpData.PositionsInRow*tmpData.PositionsInColumn;	
		 
	eTcaCarrierLayout.Layout4 :
		 tmpOffset := -0.5;
		 tmpOddRow := tmpData.PositionsInRow;
         tmpEvenRow := tmpData.PositionsInRow + 1;
         tmpWorkpieceCount := tmpData.PositionsInRow*tmpData.PositionsInColumn + tmpData.PositionsInColumn/2;
		
	eTcaCarrierLayout.Layout5 :
		 tmpOffset := 0.5;
		 tmpOddRow := tmpData.PositionsInRow;
         tmpEvenRow := tmpData.PositionsInRow - 1;
         tmpWorkpieceCount := tmpData.PositionsInRow*tmpData.PositionsInColumn - tmpData.PositionsInColumn/2;
		 
END_CASE


MEMSET(ADR(_data.WorkpiecesCoordinate),0,SIZEOF(_data.WorkpiecesCoordinate));
MEMSET(ADR(_data.WorkpiecesEnabled),0,SIZEOF(_data.WorkpiecesEnabled));


FOR ni:= 0 TO tmpWorkpieceCount-1 DO
	
	// Bestimmen des Reihen und Spaltenndex und der x und y-Koordinate
	tmpPos := ni MOD tmpWorkpieceCount;
	tmpRow := tmpPos/(tmpOddRow + tmpEvenRow);	
	tmpLoc := tmpPos MOD (tmpOddRow + tmpEvenRow);
	
	IF tmpLoc >= tmpOddRow THEN
	    // gerade Reihe
	    nRowNumber := tmpRow*2 + 1;
	    nLocationNumber := tmpLoc - tmpOddRow;
	    tmpCoordinate.fX := tmpData.ColumnDistance*(nLocationNumber + tmpOffset)+tmpData.CoordinateFirstWorkpiece.fX;
	    tmpCoordinate.fY := tmpData.RowDistance*nRowNumber+tmpData.CoordinateFirstWorkpiece.fY;
	ELSE
	    // ungerade Reihe
	    nRowNumber := tmpRow*2;
	    nLocationNumber := tmpLoc;
	    tmpCoordinate.fX := tmpData.ColumnDistance*nLocationNumber+tmpData.CoordinateFirstWorkpiece.fX;
	    tmpCoordinate.fY := tmpData.RowDistance*nRowNumber+tmpData.CoordinateFirstWorkpiece.fY;
	END_IF
	
	tmpCoordinate.nOriginId := 0;
		
	_data.WorkpiecesCoordinate[ni] := tmpCoordinate;
	_data.WorkpiecesEnabled[ni] := TRUE;

END_FOR
END_METHOD

METHOD ChangeData : ITcoTaskStatus 
VAR_INPUT
	inData : TcaCarrierData;
END_VAR
ChangeData := _ModifyTask.InvokeCarrierData(inData);
END_METHOD

METHOD ColumnDistance : REFERENCE TO TcaCarrier
VAR_INPUT
	inDistance : LREAL;
END_VAR
THIS^._config.ColumnDistance:= inDistance;
ColumnDistance REF= THIS^;
END_METHOD

METHOD CoordinateFirstWorkpiece : REFERENCE TO TcaCarrier
VAR_INPUT
	inCoordinate : ST_Coordinate;
END_VAR
THIS^._config.CoordinateFirstWorkpiece:= inCoordinate;
CoordinateFirstWorkpiece REF= THIS^;
END_METHOD

METHOD CoordinatesOf : ST_Coordinate
VAR_INPUT
	WorkpiecePlace		: INT;
END_VAR

VAR
	tmpData				: TcaCarrierConfig;
	
	tmpOffset 			: REAL;
	tmpOddRow			: INT;
	tmpEvenRow			: INT;
	tmpWorkpieceCount	: INT;
	
	tmpPos		 		: INT;
	tmpLoc		 		: INT;		
	tmpRow 				: INT;
	//tmpLvl				: INT;
	
	nRowNumber			: INT;
	nLocationNumber		: INT; 
	
	tmpCoordinate 		: ST_Coordinate;		
	
END_VAR
IF WorkpiecePlace = 0 THEN
	RETURN;
END_IF

tmpData := _config;

CASE tmpData.Layout OF
	eTcaCarrierLayout.Layout1 : 
		tmpOffset := 0;
		tmpOddRow := tmpData.PositionsInRow;
        tmpEvenRow := tmpData.PositionsInRow;
        tmpWorkpieceCount := tmpData.PositionsInRow*tmpData.PositionsInColumn;
		
    eTcaCarrierLayout.Layout2 :
		tmpOffset := 0.5;
		tmpOddRow := tmpData.PositionsInRow;
		tmpEvenRow := tmpData.PositionsInRow;
        tmpWorkpieceCount := tmpData.PositionsInRow*tmpData.PositionsInColumn;
		 
    eTcaCarrierLayout.Layout3 :
		 tmpOffset := -0.5;
		 tmpOddRow := tmpData.PositionsInRow;
         tmpEvenRow := tmpData.PositionsInRow;
         tmpWorkpieceCount := tmpData.PositionsInRow*tmpData.PositionsInColumn;	
		 
	eTcaCarrierLayout.Layout4 :
		 tmpOffset := -0.5;
		 tmpOddRow := tmpData.PositionsInRow;
         tmpEvenRow := tmpData.PositionsInRow + 1;
         tmpWorkpieceCount := tmpData.PositionsInRow*tmpData.PositionsInColumn + tmpData.PositionsInColumn/2;
		
	eTcaCarrierLayout.Layout5 :
		 tmpOffset := 0.5;
		 tmpOddRow := tmpData.PositionsInRow;
         tmpEvenRow := tmpData.PositionsInRow - 1;
         tmpWorkpieceCount := tmpData.PositionsInRow*tmpData.PositionsInColumn - tmpData.PositionsInColumn/2;
		 
END_CASE

// Bestimmen des Reihen und Spaltenndex und der x und y-Koordinate
tmpPos := (WorkpiecePlace - 1) MOD tmpWorkpieceCount;
tmpRow := tmpPos/(tmpOddRow + tmpEvenRow);	
tmpLoc := tmpPos MOD (tmpOddRow + tmpEvenRow);
//tmpLvl := (Position - 1)/tmpWorkpieceCount;


IF tmpLoc >= tmpOddRow THEN
    // gerade Reihe
    nRowNumber := tmpRow*2 + 1;
    nLocationNumber := tmpLoc - tmpOddRow;
    tmpCoordinate.fX := tmpData.ColumnDistance*(nLocationNumber + tmpOffset);
    tmpCoordinate.fY := tmpData.RowDistance*nRowNumber;
ELSE
    // ungerade Reihe
    nRowNumber := tmpRow*2;
    nLocationNumber := tmpLoc;
    tmpCoordinate.fX := tmpData.ColumnDistance*nLocationNumber;
    tmpCoordinate.fY := tmpData.RowDistance*nRowNumber;
END_IF
		

//tmpCoordinate.fZ := tmpLvl*fLevelDistance;

// Koordinaten zurückgeben
tmpCoordinate.nOriginId := 0;
CoordinatesOf := tmpCoordinate;
END_METHOD

METHOD CountEmptyPlaces : INT

VAR
	tmp				: INT;
	ni				: INT;
END_VAR
CountEmptyPlaces := 0;

FOR ni := 0 TO MAX_WORKPIECEPLACES DO
	
	IF NOT _arrayOfWorkpiecePlaces[ni].Enabled THEN
		CONTINUE;
	END_IF
	
	IF _arrayOfWorkpiecePlaces[ni].Error THEN
		CONTINUE;
	END_IF

	IF NOT _arrayOfWorkpiecePlaces[ni].WorkpiecePresent THEN
		tmp := tmp + 1;	
	END_IF

END_FOR

CountEmptyPlaces := tmp;
END_METHOD

METHOD CountPlacesByStatus : INT
VAR_INPUT
	nStatus			: INT;
END_VAR

VAR
	tmp				: INT;
	ni				: INT;
END_VAR
CountPlacesByStatus := 0;

FOR ni := 0 TO MAX_WORKPIECEPLACES DO

	IF NOT _data.WorkpiecesData[ni].Enabled THEN
		CONTINUE;
	END_IF	
	
	IF _data.WorkpiecesData[ni].Error THEN
		CONTINUE;
	END_IF

	IF _data.WorkpiecesData[ni].CurrentStatus = nStatus THEN
			tmp := tmp + 1;
	END_IF
	
END_FOR

CountPlacesByStatus := tmp;
END_METHOD

PROPERTY Data : REFERENCE TO TcaCarrierData
GET
Data REF= _data;
END_GET
END_PROPERTY

//FB_Init ist immer implizit verfügbar und wird primär für die Initialisierung verwendet.
//Der Rückgabewert wird nicht ausgewertet. Für gezielte Einflussnahme können Sie
//die Methoden explizit deklarieren und darin mit dem Standard-Initialisierungscode 
//zusätzlichen Code bereitstellen. Sie können den Rückgabewert auswerten.
METHOD FB_Init: BOOL
VAR_INPUT    
bInitRetains: BOOL; // TRUE: Die Retain-Variablen werden initialisiert (Reset warm / Reset kalt)    
bInCopyCode: BOOL;  // TRUE: Die Instanz wird danach in den Kopiercode kopiert (Online-Change)
ParentObject : ITcoObject;
END_VAR
VAR
	_i : INT;
END_VAR
FOR _i:= 0 TO MAX_WORKPIECEPLACES DO
	_arrayOfWorkpiecePlaces[_i].Id := _i+1;
END_FOR

RETURN;
END_METHOD

METHOD FillWithWorkpieces_CustomStatus : ITcoTaskStatus
VAR_INPUT
	Status		: eTcaWorkpiecePlaceStatus;
END_VAR
FillWithWorkpieces_CustomStatus := _ModifyTask.InvokeWorkpieceCommand(eTcaCarrierCmd.fillPlaces, Status);
END_METHOD

METHOD FillWithWorkpieces_InitialStatus : ITcoTaskStatus
VAR_INPUT
END_VAR
IF _data.RequestStatus = eTcaWorkpiecePlaceStatus.undefined THEN
	RETURN;
END_IF

FillWithWorkpieces_InitialStatus := _ModifyTask.InvokeWorkpieceCommand(eTcaCarrierCmd.fillPlaces, _data.InitialStatus);
END_METHOD

{attribute 'TcRpcEnable'}
METHOD FillWithWorkpieces_RequestStatus : ITcoTaskStatus
VAR_INPUT
END_VAR
IF Data.RequestStatus = eTcaWorkpiecePlaceStatus.undefined THEN
	RETURN;
END_IF

FillWithWorkpieces_RequestStatus := _ModifyTask.InvokeWorkpieceCommand(eTcaCarrierCmd.fillPlaces, Data.RequestStatus);
END_METHOD

METHOD FindPlace : REFERENCE TO TcaWorkpiecePlace //-1..no Position found

VAR_INPUT
	Status		: eTcaWorkpiecePlaceStatus;
END_VAR

VAR
	ni				: INT;
END_VAR
FindPlace REF= 0;
FOR ni := 0 TO MAX_WORKPIECEPLACES DO
	
	IF NOT _data.WorkpiecesData[ni].Enabled THEN
		CONTINUE;
	END_IF	
	
	IF _data.WorkpiecesData[ni].Error THEN
		CONTINUE;
	END_IF	

	IF _data.WorkpiecesData[ni].CurrentStatus = Status OR Status < eTcaWorkpiecePlaceStatus.undefined THEN
	   
		FindPlace REF= _arrayOfWorkpiecePlaces[ni];
		EXIT;
		
	END_IF	
END_FOR
END_METHOD

METHOD GetPlaceReference : REFERENCE TO TcaWorkpiecePlace
VAR_INPUT
	nIndexNr		: INT;
END_VAR
IF nIndexNr < 0 OR nIndexNr > MAX_WORKPIECEPLACES THEN
	RETURN;
END_IF

GetPlaceReference REF= _arrayOfWorkpiecePlaces[nIndexNr];
END_METHOD

PROPERTY InitialStatus : eTcaWorkpiecePlaceStatus
GET
InitialStatus := _data.InitialStatus;
END_GET
SET
_data.InitialStatus := InitialStatus;
END_SET
END_PROPERTY

METHOD Layout : REFERENCE TO TcaCarrier
VAR_INPUT
	inLayout : eTcaCarrierLayout;
END_VAR
THIS^._config.Layout:= inLayout;
Layout REF= THIS^;
END_METHOD

PROPERTY ModifyTask : TcoCore.ITcoTaskStatus
GET
ModifyTask := _ModifyTask;
END_GET
END_PROPERTY

METHOD PositionsInColumn : REFERENCE TO TcaCarrier
VAR_INPUT
	inPositionsInColumn : INT;
END_VAR
THIS^._config.PositionsInColumn:= inPositionsInColumn;
PositionsInColumn REF= THIS^;
END_METHOD

METHOD PositionsInRow : REFERENCE TO TcaCarrier
VAR_INPUT
	inPositionsInRow : INT;
END_VAR
THIS^._config.PositionsInRow:= inPositionsInRow;
PositionsInRow REF= THIS^;
END_METHOD

METHOD RefreshStatus : BOOL
VAR
	ni			: INT;
END_VAR
MEMSET(ADR(_WorkpieceStatusCount), 0, SIZEOF(_WorkpieceStatusCount));
_data.InitialStatus := eTcaWorkpiecePlaceStatus.undefined;
_data.RequestStatus := eTcaWorkpiecePlaceStatus.undefined;

FOR ni := 0 TO MAX_WORKPIECEPLACES DO
	
	IF NOT _arrayOfWorkpiecePlaces[ni].Enabled THEN
		CONTINUE;
	END_IF

		
	IF _data.WorkpiecesData[ni].CurrentStatus = eTcaWorkpiecePlaceStatus.undefined THEN
		CONTINUE;
	END_IF

	_WorkpieceStatusCount[_data.WorkpiecesData[ni].CurrentStatus] := _WorkpieceStatusCount[_data.WorkpiecesData[ni].CurrentStatus] + 1;
	
	IF _WorkpieceStatusCount[_data.WorkpiecesData[ni].CurrentStatus] >= _WorkpieceStatusCount[_PrimaryStatus] THEN
		_SecondaryStatus := _PrimaryStatus;
		_PrimaryStatus := _data.WorkpiecesData[ni].CurrentStatus;
	END_IF

END_FOR


IF _PrimaryStatus = _SecondaryStatus THEN
	_SecondaryStatus := 0;
END_IF

_modifyId := _modifyId + 1;
END_METHOD

PROPERTY RequestStatus : eTcaWorkpiecePlaceStatus
GET
RequestStatus := _data.RequestStatus;
END_GET
SET
_data.RequestStatus := RequestStatus;
END_SET
END_PROPERTY

(*~
	<docu>
		<summary>
			Restores this instance to the Ready state. Can be called explicitly or from within one of the restore mechanisms.	
		</summary>			
	</docu>	
~*)
METHOD Restore : TcoCore.ITcoRestorable

VAR
	_i : INT;
END_VAR
FOR _i:= 0 TO MAX_WORKPIECEPLACES DO
	_arrayOfWorkpiecePlaces[_i].Restore();
END_FOR

RefreshStatus();
END_METHOD

METHOD RowDistance : REFERENCE TO TcaCarrier
VAR_INPUT
	inDistance : LREAL;
END_VAR
THIS^._config.RowDistance:= inDistance;
RowDistance REF= THIS^;
END_METHOD

(*~
	<docu>
		<summary>
		    Custom service (manual, maintenance) logic.
			This method must be implemented in derived class.
		</summary>			
	</docu>	
~*)
METHOD PROTECTED ServiceMode
VAR
	_i : INT;
END_VAR
FOR _i:= 0 TO MAX_WORKPIECEPLACES DO
	_arrayOfWorkpiecePlaces[_i].Service();
END_FOR
END_METHOD

PROPERTY Task : TcoCore.ITcoTask
GET
Task := _ModifyTask;
END_GET
END_PROPERTY

PROPERTY WorkpiecePlaces : INT
GET
CASE _config.Layout OF	
	eTcaCarrierLayout.Layout1 : WorkpiecePlaces := _config.PositionsInRow*_config.PositionsInColumn;		
    eTcaCarrierLayout.Layout2 : WorkpiecePlaces := _config.PositionsInRow*_config.PositionsInColumn;		 
    eTcaCarrierLayout.Layout3 : WorkpiecePlaces := _config.PositionsInRow*_config.PositionsInColumn;		 
	eTcaCarrierLayout.Layout4 : WorkpiecePlaces := _config.PositionsInRow*_config.PositionsInColumn + _config.PositionsInColumn/2;		
	eTcaCarrierLayout.Layout5 : WorkpiecePlaces := _config.PositionsInRow*_config.PositionsInColumn - _config.PositionsInColumn/2;		
	ELSE
		 WorkpiecePlaces := 0;
END_CASE
END_GET
END_PROPERTY

END_FUNCTION_BLOCK

// ---- Components/TcaCarrier/Tasks/TcaCarrierModifyTask.TcPOU
FUNCTION_BLOCK TcaCarrierModifyTask EXTENDS TcoCore.TcoTask



VAR_IN_OUT
	inoArrayOfWorkpiecePlaces : ARRAY[*] OF TcaWorkpiecePlace(THIS^);	
END_VAR
VAR
	_Command : eTcaCarrierCmd;
	_StatusOfPlace : eTcaWorkpiecePlaceStatus;
	_CarrierData : TcaCarrierData;
END_VAR
VAR
    {attribute 'hide'}
	_WorkpiecePlaces : INT;
    {attribute 'hide'}
	_i	: DINT;
END_VAR

IF(Execute()) THEN	
	
	// Change of Config -> set to empty Place
	IF _Command = eTcaCarrierCmd.ConfigCarrier THEN
		Carrier.Data := _CarrierData;
		_Command := eTcaCarrierCmd.emptyPlaces;
		_StatusOfPlace := eTcaWorkpiecePlaceStatus.undefined;
	END_IF
	
	Carrier.RefreshStatus();
	
	IF Carrier.WorkpiecePlaces = 0 THEN
		RETURN;
	END_IF

	CASE _Command OF	

	eTcaCarrierCmd.emptyPlaces : 
		FOR _i := LOWER_BOUND(inoArrayOfWorkpiecePlaces,1) TO UPPER_BOUND(inoArrayOfWorkpiecePlaces,1) DO
			inoArrayOfWorkpiecePlaces[_i].Restore();
			inoArrayOfWorkpiecePlaces[_i].Data.CurrentStatus := _StatusOfPlace;
			inoArrayOfWorkpiecePlaces[_i].Enabled := TRUE;
			inoArrayOfWorkpiecePlaces[_i].Id := TO_INT(_i)+1;
		END_FOR
		
		FOR _i := _WorkpiecePlaces TO UPPER_BOUND(inoArrayOfWorkpiecePlaces,1) DO
			inoArrayOfWorkpiecePlaces[_i].Restore();
			inoArrayOfWorkpiecePlaces[_i].Data.CurrentStatus := eTcaWorkpiecePlaceStatus.undefined;
			inoArrayOfWorkpiecePlaces[_i].Enabled := FALSE;
			inoArrayOfWorkpiecePlaces[_i].Id := -1;
		END_FOR
			

	eTcaCarrierCmd.fillPlaces : 
		FOR _i := LOWER_BOUND(inoArrayOfWorkpiecePlaces,1) TO _WorkpiecePlaces-1 DO
			inoArrayOfWorkpiecePlaces[_i].Data.CurrentStatus := _StatusOfPlace;
			inoArrayOfWorkpiecePlaces[_i].Enabled := TRUE;
			inoArrayOfWorkpiecePlaces[_i].Id := TO_INT(_i)+1;
		END_FOR
		
		FOR _i := _WorkpiecePlaces TO UPPER_BOUND(inoArrayOfWorkpiecePlaces,1) DO
			inoArrayOfWorkpiecePlaces[_i].Restore();
			inoArrayOfWorkpiecePlaces[_i].Data.CurrentStatus := eTcaWorkpiecePlaceStatus.undefined;
			//inoArrayOfWorkpiecePlaces[_i].Id := -1;
		END_FOR
	
	eTcaCarrierCmd.RestorePlaces : 
		FOR _i := LOWER_BOUND(inoArrayOfWorkpiecePlaces,1) TO UPPER_BOUND(inoArrayOfWorkpiecePlaces,1) DO
			inoArrayOfWorkpiecePlaces[_i].Restore();
			//inoArrayOfWorkpiecePlaces[_i].Id := -1;
			inoArrayOfWorkpiecePlaces[_i].Data.CurrentStatus := eTcaWorkpiecePlaceStatus.undefined;
		END_FOR

	END_CASE
	
	Carrier.RefreshStatus();
	DoneWhen(TRUE);
	Restore();
END_IF

PROPERTY Carrier : REFERENCE TO TcaCarrier
GET
VAR
    _carrier : POINTER TO TcaCarrier;
END_VAR
IF __QUERYPOINTER(_ParentObject,_carrier) THEN 	// Check if _Parent is Carrier
	Carrier REF= _carrier^;              		// If the check is successful dereference a pointer. simlar to THIS^ or SUPER^
END_IF
END_GET
END_PROPERTY

METHOD InvokeCarrierData : ITcoTaskStatus
VAR_INPUT
	inData : TcaCarrierData;
END_VAR
_CarrierData := inData;
InvokeCarrierData := This^.Invoke();
END_METHOD

METHOD InvokeWorkpieceCommand : ITcoTaskStatus
VAR_INPUT
	inCommand : eTcaCarrierCmd;
	inStatusOfWorkpiece : eTcaWorkpiecePlaceStatus;
END_VAR
_Command := inCommand;
_StatusOfPlace := inStatusOfWorkpiece;
InvokeWorkpieceCommand := This^.Invoke();
END_METHOD

END_FUNCTION_BLOCK

// ---- Components/TcaStorage/TcaStorage.TcPOU
FUNCTION_BLOCK TcaStorage EXTENDS TcoCore.TcoComponent

VAR_INPUT
	ref : REFERENCE TO TcaStorageRef;
END_VAR

VAR	
	_Dock : BOOL;
	_Carrier : TcaCarrier(THIS^);
	_CarrierSensor : TcoDi(THIS^);	
	_CarrierPresent : BOOL;

	_Task : TcoCore.TcoTask(THIS^);	
	_cmd : eTcaStorageCmd;
	
	// Carrier Setting
	fbCarrierTemplate	: TcaCarrier(THIS^);	

END_VAR

IF NOT __ISVALIDREF(ref) THEN
	_Dock := FALSE;
ELSE
	_Dock := TRUE;
	_CarrierSensor(inoSignal := ref.Sensor);
END_IF


IF _Task.Done THEN
	_Task.Restore();
END_IF


IF _Task.Execute() THEN
	RETURN;
END_IF


CASE _cmd OF
	
	eTcaStorageCmd.FillCarrier:
		AddCarrier().FillWithWorkpieces_InitialStatus();
			
	eTcaStorageCmd.RemoveCarrier:
		RemoveCarrier();
	
	eTcaStorageCmd.EmptyCarrier:
		;
	
END_CASE
	

_Task.DoneWhen(TRUE);

METHOD AddCarrier : REFERENCE TO TcaCarrier
_CarrierPresent := TRUE;
_Carrier.Restore();
AddCarrier REF= _Carrier;
END_METHOD

PROPERTY CarrierPresent : BOOL
GET
CarrierPresent := _CarrierSensor.Signal;
END_GET
END_PROPERTY

METHOD RemoveCarrier : REFERENCE TO TcaCarrier
VAR
END_VAR
_CarrierPresent := FALSE;
_Carrier.Restore();
RemoveCarrier REF= _Carrier;
END_METHOD

(*~
	<docu>
		<summary>
			Restores this instance to the Ready state. Can be called explicitly or from within one of the restore mechanisms.	
		</summary>			
	</docu>	
~*)
METHOD Restore : TcoCore.ITcoRestorable
END_METHOD

(*~
	<docu>
		<summary>
		    Custom service (manual, maintenance) logic.
			This method must be implemented in derived class.
		</summary>			
	</docu>	
~*)
METHOD PROTECTED ServiceMode
_Carrier.Service();
END_METHOD

END_FUNCTION_BLOCK

// ---- Components/TcaTrolley/TcaTrolley.TcPOU
FUNCTION_BLOCK TcaTrolley EXTENDS TcoCore.TcoComponent

VAR CONSTANT
	MAX_CARRIERPLACES : INT := 63;
END_VAR


VAR PERSISTENT
	_data : TcaTrolleyData;
END_VAR

PROPERTY Data : REFERENCE TO TcaTrolleyData
GET
Data REF= _data;
END_GET
SET
_data := Data;
END_SET
END_PROPERTY

{warning 'Methodenimplementierung hinzufügen'}
METHOD Restore : TcoCore.ITcoRestorable
END_METHOD

{warning 'Methodenimplementierung hinzufügen'}
(*~
	<docu>
		<summary>
		    Custom service (manual, maintenance) logic.
			This method must be implemented in derived class.
		</summary>			
	</docu>	
~*)
METHOD PROTECTED ServiceMode
END_METHOD

END_FUNCTION_BLOCK

// ---- Components/TcaPushButton/TcaPushButton.TcPOU
FUNCTION_BLOCK TcaPushButton EXTENDS TcoCore.TcoComponent

VAR_INPUT
	ref : REFERENCE TO TcaPushButtonRef;
END_VAR

VAR
	_status : TcaPushButtonStatus;
	_config : TcaPushButtonConfig;
	_service : TcaPushButtonService;
	
	_tonSignal : TON;
	_rtSignal : R_TRIG;
	_ftSignal : F_TRIG;
	
    _LightTask : TcoCore.TcoTask(THIS^);	
	_FlashArrayId : INT;
	
END_VAR

IF NOT __ISVALIDREF(ref)  THEN
    Messenger.Post('<#Invalid reference signal #>', TcoCore.eMessageCategory.ProgrammingError);
    RETURN;
END_IF

// Signal Postprocessing
_tonSignal(IN:= ref.Button , PT:= _config.ValidationTime);
_rtSignal(CLK:= _tonSignal.Q OR _service.Button, Q=>);
_ftSignal(CLK:= _tonSignal.Q OR _service.Button, Q=>);

// Task
_lighttask.Enabled := TRUE;
IF NOT (_lighttask.Execute()) THEN
	RETURN;
END_IF
	
CASE _status.LightState OF 
	
eTcaPushButtonLightState.none:
	ref.Light := FALSE;

eTcaPushButtonLightState.permanent:
	ref.Light := TRUE;

eTcaPushButtonLightState.intervall:
	IF _lighttask.ElapsedTime > _config.FlashArray[_FlashArrayId] THEN
		ref.Light := (_FlashArrayId MOD 2 <> 0);	
		_FlashArrayId := _FlashArrayId + 1;
	END_IF
	
	IF _config.FlashArray[_FlashArrayId] = T#0MS THEN
		_FlashArrayId := 0;
		_lighttask.Restore();
		_lighttask.Invoke();
	END_IF	
	
END_CASE

// Refresh Status
_status.Light := ref.Light;
_status.Falling := _ftSignal.Q;
_status.Raising := _rtSignal.Q;
_status.Signal := _tonSignal.Q;
_status.ElapsedTime :=  _tonSignal.ET;
THIS^.Status;

METHOD Blink : ITcoTaskStatus
VAR_INPUT
	BlinkIntervall : TIME;
END_VAR
MEMSET(ADR(_config.FlashArray), 0, SIZEOF(_config.FlashArray));

_config.FlashArray[0] := BlinkIntervall;
_config.FlashArray[1] := BlinkIntervall*2;

IF _status.LightState <> eTcaPushButtonLightState.Intervall THEN
	_status.LightState := eTcaPushButtonLightState.Intervall;
	Blink := _LightTask.Invoke();
END_IF
END_METHOD

PROPERTY Config : REFERENCE TO TcaPushButtonConfig
GET
Config Ref= _config;
END_GET
SET
_config := Config;
END_SET
END_PROPERTY

METHOD Flash : ITcoTaskStatus
VAR_INPUT
	FlashCount : INT;
END_VAR

VAR
	_BlinkIntervall : TIME := T#1000MS;
	_FlashIntervall : TIME := T#200MS;
	_Count : INT;
END_VAR
MEMSET(ADR(_config.FlashArray), 0, SIZEOF(_config.FlashArray));

_config.FlashArray[0] := _BlinkIntervall;
_config.FlashArray[1] := _BlinkIntervall*2;

FOR _Count := 0 TO 2*FlashCount BY 2 DO
	_config.FlashArray[2+_Count] := _FlashIntervall + _config.FlashArray[1+_Count];
	_config.FlashArray[3+_Count] := _FlashIntervall + _config.FlashArray[2+_Count];
END_FOR

IF _status.LightState <> eTcaPushButtonLightState.Intervall THEN
	_status.LightState := eTcaPushButtonLightState.Intervall;
	Flash := _LightTask.Invoke();
END_IF
END_METHOD

PROPERTY LightTask : TcoCore.ITcoTask
GET
LightTask := _LightTask;
END_GET
END_PROPERTY

METHOD Off : ITcoTaskStatus
VAR_INPUT
END_VAR
IF _status.LightState <> eTcaPushButtonLightState.none THEN
	_status.LightState := eTcaPushButtonLightState.none;
	Off := _LightTask.Invoke();
END_IF
END_METHOD

METHOD On : ITcoTaskStatus
VAR_INPUT
END_VAR
IF _status.LightState <> eTcaPushButtonLightState.permanent THEN
	_status.LightState := eTcaPushButtonLightState.permanent;
	On := _LightTask.Invoke();
END_IF
END_METHOD

{warning 'Methodenimplementierung hinzufügen'}
METHOD Restore : TcoCore.ITcoRestorable
END_METHOD

{warning 'Methodenimplementierung hinzufügen'}
(*~
	<docu>
		<summary>
		    Custom service (manual, maintenance) logic.
			This method must be implemented in derived class.
		</summary>			
	</docu>	
~*)
METHOD PROTECTED ServiceMode
END_METHOD

PROPERTY Status : REFERENCE TO TcaPushButtonStatus
GET
Status REF= _status;

_service.Light := _status.Light;
END_GET
END_PROPERTY

END_FUNCTION_BLOCK

// ---- Components/TcaTrolley_old/TcaTrolley_old.TcPOU
FUNCTION_BLOCK TcaTrolley_old EXTENDS TcoCore.TcoObject

VAR CONSTANT
	nMaxWorkpieceCarrier : INT := 31;
END_VAR

VAR_INPUT
	ref : REFERENCE TO TcaTrolleyRef;
END_VAR

VAR
	
	bDock					: BOOL;
	fbTrolleyPresent		: TcoDi(THIS^);	
	bTrolleyPresent			: BOOL;
	
	
	// Trolley Setting	
	nStoragePerRack			: INT;
	fStorageDivision		: LREAL;
	stOrigin				: ST_Coordinate; //mirrored for the Right side
	
	// Carrier Setting	
	fbCarrierTemplate		: TcaCarrier_(THIS^);	
	
END_VAR

VAR_OUTPUT PERSISTENT
	aLeftRack				: ARRAY[0..nMaxWorkpieceCarrier] OF TcaWorkpieceCarrier(THIS^);
	aRightRack				: ARRAY[0..nMaxWorkpieceCarrier] OF TcaWorkpieceCarrier(THIS^);
	bLeftRackPresent		: ARRAY[0..nMaxWorkpieceCarrier] OF BOOL;	
	bRightRackPresent		: ARRAY[0..nMaxWorkpieceCarrier] OF BOOL;	
END_VAR

VAR_INPUT
	cmd						: CMD_Trolley;
END_VAR

IF NOT __ISVALIDREF(ref) THEN
	bDock := FALSE;
ELSE
	bDock := TRUE;
	fbTrolleyPresent(inoSignal := ref.Sensor);
END_IF

METHOD AddCarrier : TcoCore.ITcoTaskStatus
VAR_IN_OUT
	WorkpieceCarrier			: TcaWorkpieceCarrier;
END_VAR
VAR_INPUT	
	bLeft						: BOOL;
	bRight						: BOOL;
	nId							: INT;
END_VAR
IF bLeft THEN
	MEMCPY(ADR(aLeftRack[nId]), ADR(WorkpieceCarrier), SIZEOF(TcaWorkpieceCarrier));
	bLeftRackPresent[nId] := TRUE;	
	aLeftRack[nId].RefreshCounter();
END_IF

IF bRight THEN
	MEMCPY(ADR(aRightRack[nId]), ADR(WorkpieceCarrier), SIZEOF(TcaWorkpieceCarrier));
	bRightRackPresent[nId] := TRUE;
	aRightRack[nId].RefreshCounter();
END_IF
END_METHOD

METHOD DefineCarrier
VAR_INPUT
	eConfiguration				: eTcaCarrierConfig;	
    nPosInRow					: INT;			// Numbers of Positions in first Row
    fRowDistance				: REAL;		// Distance from one Row to the other 
    nPosInColumn				: INT;			// Numbers of Positions in one Column
    fColumnDistance				: REAL;		// Distance from one Column to the other
END_VAR
fbCarrierTemplate.PositionInColumn :=	nPosInColumn;
fbCarrierTemplate.PositionInRow := nPosInRow;
fbCarrierTemplate.ColumnDistance := fColumnDistance;
fbCarrierTemplate.RowDistance := fRowDistance;
fbCarrierTemplate.Configuration := eConfiguration;
END_METHOD

METHOD DefineTrolley
VAR_INPUT
	StoragePerRack		: INT;
	StorageDivision		: LREAL;
	//Origin				: ST_Coordinate; //mirrored for the Right side
END_VAR
nStoragePerRack := StoragePerRack;
fStorageDivision := StorageDivision;
//stOrigin := Origin;
END_METHOD

METHOD EmptyCarrier : BOOL
VAR_INPUT
	bLeft			: BOOL;
	bRight			: BOOL;
	nState			: INT;
	nId				: INT;
END_VAR
IF bLeft THEN
	IF aLeftRack[nId].CarrierId = -1 THEN
		EmptyCarrier := TRUE;
	END_IF	

	aLeftRack[nId].LoadTemplate(fbCarrierTemplate);
	aLeftRack[nId].EmptyPlaces(nState);
	aLeftRack[nId].CarrierId := nId+1;
	aLeftRack[nId].RefreshCounter();
	bLeftRackPresent[nId] := FALSE;
END_IF

IF bRight THEN
	IF aRightRack[nId].CarrierId = -1 THEN
		EmptyCarrier := TRUE;
	END_IF	
	
	aRightRack[nId].LoadTemplate(fbCarrierTemplate);
	aRightRack[nId].EmptyPlaces(nState);
	aRightRack[nId].CarrierId := nId+1;
	aRightRack[nId].RefreshCounter();
	bRightRackPresent[nId] := FALSE;
END_IF
END_METHOD

METHOD EmptyTrolley : BOOL
VAR_INPUT
	bLeft			: BOOL;
	bRight			: BOOL;
END_VAR

VAR
	tmpNew			: BOOL;
	ni				: INT;
END_VAR
FOR ni:= 0 TO nMaxWorkpieceCarrier DO

	IF EmptyCarrier(bLeft, bRight, -1, ni) THEN
		tmpNew := TRUE;
	END_IF

END_FOR

IF tmpNew THEN
	ChangeToggle();
END_IF
END_METHOD

METHOD NewCarrier : BOOL
VAR_INPUT
	bLeft			: BOOL;
	bRight			: BOOL;
	nId				: INT;
	nState			: INT;
END_VAR
IF bLeft THEN
	IF aLeftRack[nId].CarrierId = -1 THEN
		NewCarrier := TRUE;
	END_IF

	aLeftRack[nId].LoadTemplate(fbCarrierTemplate);
	aLeftRack[nId].FillPlaces(nState);
	aLeftRack[nId].CarrierId := nId+1;
	aLeftRack[nId].RefreshCounter();
	bLeftRackPresent[nId] := TRUE;
END_IF

IF bRight THEN
	IF aRightRack[nId].CarrierId = -1 THEN
		NewCarrier := TRUE;
	END_IF	

	aRightRack[nId].LoadTemplate(fbCarrierTemplate);
	aRightRack[nId].FillPlaces(nState);
	aRightRack[nId].CarrierId := nId+1;
	aRightRack[nId].RefreshCounter();
	bRightRackPresent[nId] := TRUE;
END_IF
END_METHOD

METHOD NewTrolley : BOOL
VAR_INPUT
	bLeft			: BOOL;
	bRight			: BOOL;
	nState			: INT;
END_VAR

VAR
	tmpNew			: BOOL;
	ni				: INT;
END_VAR
FOR ni:= 0 TO nMaxWorkpieceCarrier DO

	IF NewCarrier(bLeft, bRight, ni, nState) THEN
		tmpNew := TRUE;
	END_IF
	
END_FOR

IF tmpNew THEN
	ChangeToggle();
END_IF
END_METHOD

METHOD RefreshTrolley
VAR
	ni	: INT;
END_VAR
FOR ni:= 0 TO nMaxWorkpieceCarrier DO
	aLeftRack[ni].RefreshCounter();
	aRightRack[ni].RefreshCounter();
END_FOR
END_METHOD

METHOD RemoveCarrier : TcoCore.ITcoTaskStatus
VAR_INPUT
	bLeft			: BOOL;
	bRight			: BOOL;
	nId				: INT;
END_VAR
IF bLeft THEN
	aLeftRack[nId].ResetPlaces();
	aLeftRack[nId].CarrierId := -1;
	bLeftRackPresent[nId] := FALSE;
	aLeftRack[nId].RefreshCounter();
END_IF

IF bRight THEN
	aRightRack[nId].ResetPlaces();
	aRightRack[nId].CarrierId := -1;
	bRightRackPresent[nId] := FALSE;
	aRightRack[nId].RefreshCounter();
END_IF
END_METHOD

METHOD RemoveTrolley : BOOL
VAR_INPUT
	bLeft			: BOOL;
	bRight			: BOOL;
END_VAR

VAR
	ni				: INT;
END_VAR
FOR ni:= 0 TO nMaxWorkpieceCarrier DO

	RemoveCarrier(bLeft, bRight, ni);

END_FOR

ChangeToggle();
END_METHOD

(*~
	<docu>
		<summary>
			Restores this instance to the Ready state. Can be called explicitly or from within one of the restore mechanisms.	
		</summary>			
	</docu>	
~*)
METHOD Restore : TcoCore.ITcoRestorable
END_METHOD

/// RunSuper component logic
{attribute 'object_name' := 'Run'}
METHOD  Run
END_METHOD

(*~
	<docu>
		<summary>
		    Custom service (manual, maintenance) logic.
			This method must be implemented in derived class.
		</summary>			
	</docu>	
~*)
METHOD PROTECTED ServiceMode
END_METHOD

/// Visu component logic
{attribute 'object_name' := 'Visu'}
METHOD  Visu

VAR
	ni			:INT;
END_VAR
CASE cmd.cmd OF
	eTcaTrolleyCmd.FillTrolley:
		NewTrolley(TRUE, TRUE, cmd.nId);
	
	eTcaTrolleyCmd.EmptyTrolley:
		EmptyTrolley(TRUE, TRUE);
	
	eTcaTrolleyCmd.RemoveTrolley:
		RemoveTrolley(TRUE, TRUE);
		
END_CASE

IF cmd.cmd <> eTcaTrolleyCmd.noCmd THEN
	cmd.cmd := eTcaTrolleyCmd.noCmd; 
END_IF

FOR ni:= 0 TO nMaxWorkpieceCarrier DO
	IF aLeftRack[ni].Cmd = eTcaCarrierCmd.changeState THEN
		NewCarrier(TRUE, FALSE, ni, cmd.nId);
		aLeftRack[ni].Cmd := eTcaCarrierCmd.noCmd;
	END_IF
	
	IF aRightRack[ni].Cmd = eTcaCarrierCmd.changeState THEN
		NewCarrier(FALSE, TRUE, ni, cmd.nId);
		aRightRack[ni].Cmd := eTcaCarrierCmd.noCmd;
	END_IF
	
END_FOR
END_METHOD

END_FUNCTION_BLOCK

// ---- Components_RMTH/TcaSegmentDoor/TcaSegmentDoor.TcPOU
FUNCTION_BLOCK TcaSegmentDoor EXTENDS TcoComponent

VAR_INPUT
	ref : REFERENCE TO TcaSegmentDoorRef;
END_VAR

VAR
	_status : TcaSegmentDoorStatus;
	_config : TcaSegmentDoorConfig;
	_service : TcaSegmentDoorService;
	
	//Tasks
	_closeTask : TcoCore.TcoTask(THIS^);
	_openTask : TcoCore.TcoTask(THIS^);
	_initTask : TcoCore.TcoTask(THIS^);
	
	_EnableAxis : BOOL := TRUE;
	_EnableAxisSafe : BOOL;
	
	// Components
	_vertikalAxis : TcoDriveSimple(THIS^);	
	_latchLeft : TcoDriveSimple(THIS^);
	_latchRight : TcoDriveSimple(This^);

END_VAR

IF NOT __ISVALIDREF(ref)  THEN
    Messenger.Post('<#Invalid reference signal #>', TcoCore.eMessageCategory.ProgrammingError);
    RETURN;
END_IF

// Axis
_EnableAxisSafe := _EnableAxis; //AND ref.tsSS1;
_vertikalAxis(inCalibrationCam:= ref.ReferenceSensor, inEnable:=  _EnableAxisSafe , inEnableNegative:= _EnableAxisSafe, inEnablePositive:= _EnableAxisSafe, inoAxisRef:= ref.VertikalAxis);
_latchLeft( inEnable:= _EnableAxisSafe, inEnableNegative:= _EnableAxisSafe, inEnablePositive:= _EnableAxisSafe, inoAxisRef:= ref.LatchLeft);
_latchRight( inEnable:= _EnableAxisSafe, inEnableNegative:= _EnableAxisSafe, inEnablePositive:= _EnableAxisSafe, inoAxisRef:= ref.LatchRight);

METHOD Close : ITcoTaskStatus
VAR_INPUT
END_VAR
_closeTask.Restore();
Close := _closeTask.Invoke();
END_METHOD

PROPERTY CloseTask : TcoCore.ITcoTask
GET
CloseTask := _CloseTask;
END_GET
END_PROPERTY

PROPERTY Config : REFERENCE TO TcaSegmentDoorConfig
GET
Config Ref= _config;
END_GET
SET
_config := Config;
END_SET
END_PROPERTY

